# B&R Automation Studio project NAINV104C00R8L515F00 (part 11)

#### Act_OptP0200ToP0201AccDat.st
```iecst
ACTION Act_OptP0200ToP0201AccDat:

	//Control
	IF (tyP0200OpsGen.tyOps.tyBtnAccDat.bRtCompl = TRUE) OR (tyP0201OpsConv.tyOps.tyBtnAccDat.bRtCompl = TRUE) THEN
		tyP0200OpsGen.tyOps.tyBtnAccDat.bRtCompl	:= FALSE;
		tyP0201OpsConv.tyOps.tyBtnAccDat.bRtCompl	:= FALSE;

		bProdAccData	:= TRUE;
	END_IF

	//Button Appearance
	IF (p_bLFFollowerProdAccDataMnl = TRUE) OR (p_bUSHermesAccDataMnl = TRUE) OR (p_bLCSLFAccDataMnl = TRUE) THEN

		fbAccDatBlinkTm(IN := TRUE);

		IF fbAccDatBlinkTm.Q THEN
			fbAccDatBlinkTm(IN := FALSE);
			IF tyP0200OpsGen.tyOps.tyBitmapAccDat.usiValueIdx = 1 THEN
				tyP0200OpsGen.tyOps.tyBitmapAccDat.usiValueIdx		:= 0;
				tyP0201OpsConv.tyOps.tyBitmapAccDat.usiValueIdx	:= 0;
			ELSE
				tyP0200OpsGen.tyOps.tyBitmapAccDat.usiValueIdx		:= 1;
				tyP0201OpsConv.tyOps.tyBitmapAccDat.usiValueIdx	:= 1;
			END_IF
		END_IF

		fUIInRtStatOff(ADR(tyP0200OpsGen.tyOps.tyBtnAccDat.uiRtStat));
		fUIInRtStatOff(ADR(tyP0201OpsConv.tyOps.tyBtnAccDat.uiRtStat));

		fUIInRtStatOff(ADR(tyP0200OpsGen.tyOps.tyBitmapAccDat.uiRtStat));
		fUIInRtStatOff(ADR(tyP0201OpsConv.tyOps.tyBitmapAccDat.uiRtStat));

	ELSE

		fbAccDatBlinkTm(IN := FALSE);

		tyP0200OpsGen.tyOps.tyBitmapAccDat.usiValueIdx	:= 0;
		tyP0201OpsConv.tyOps.tyBitmapAccDat.usiValueIdx	:= 0;

		fUIInRtStatHide(ADR(tyP0200OpsGen.tyOps.tyBtnAccDat.uiRtStat));
		fUIInRtStatHide(ADR(tyP0201OpsConv.tyOps.tyBtnAccDat.uiRtStat));

		fUIInRtStatHide(ADR(tyP0200OpsGen.tyOps.tyBitmapAccDat.uiRtStat));
		fUIInRtStatHide(ADR(tyP0201OpsConv.tyOps.tyBitmapAccDat.uiRtStat));

	END_IF

//	IF p_tyNtParamCurr.bLFPrep THEN
//		IF p_bLFFollowerDSAllow=FALSE THEN
//			tyP0200OpsGen.tyOps.tyTxtLdrInActiveCtrl.usiValueIdx	:= 0;
//			tyP0201OpsConv.tyOps.tyTxtLdrInActiveCtrl.usiValueIdx	:= 0;
//
//			fUIInRtStatOff(ADR(tyP0200OpsGen.tyOps.tyTxtLdrInActiveCtrl.uiRtStat));
//			fUIInRtStatOff(ADR(tyP0201OpsConv.tyOps.tyTxtLdrInActiveCtrl.uiRtStat));
//			fUIInRtStatOff(ADR(tyP0200OpsGen.tyOps.tyBitmapWarningLF.uiRtStat));
//			fUIInRtStatOff(ADR(tyP0201OpsConv.tyOps.tyBitmapWarningLF.uiRtStat));
//
//		ELSIF p_bLFFollowerUSAllow=FALSE THEN
//			IF p_tyMcParamCurr.bSectionLeader THEN
//				tyP0200OpsGen.tyOps.tyTxtLdrInActiveCtrl.usiValueIdx	:= 3;
//				tyP0201OpsConv.tyOps.tyTxtLdrInActiveCtrl.usiValueIdx	:= 3;
//
//				fUIInRtStatOff(ADR(tyP0200OpsGen.tyOps.tyTxtLdrInActiveCtrl.uiRtStat));
//				fUIInRtStatOff(ADR(tyP0201OpsConv.tyOps.tyTxtLdrInActiveCtrl.uiRtStat));
//				fUIInRtStatOff(ADR(tyP0200OpsGen.tyOps.tyBitmapWarningLF.uiRtStat));
//				fUIInRtStatOff(ADR(tyP0201OpsConv.tyOps.tyBitmapWarningLF.uiRtStat));
//			ELSE
//				tyP0200OpsGen.tyOps.tyTxtLdrInActiveCtrl.usiValueIdx	:= 2;
//				tyP0201OpsConv.tyOps.tyTxtLdrInActiveCtrl.usiValueIdx	:= 2;
//
//				fUIInRtStatOff(ADR(tyP0200OpsGen.tyOps.tyTxtLdrInActiveCtrl.uiRtStat));
//				fUIInRtStatOff(ADR(tyP0201OpsConv.tyOps.tyTxtLdrInActiveCtrl.uiRtStat));
//				fUIInRtStatOff(ADR(tyP0200OpsGen.tyOps.tyBitmapWarningLF.uiRtStat));
//				fUIInRtStatOff(ADR(tyP0201OpsConv.tyOps.tyBitmapWarningLF.uiRtStat));
//			END_IF
//		ELSE
//			IF p_bLFFollowerLdrSeqCtrlInActive THEN
//				tyP0200OpsGen.tyOps.tyTxtLdrInActiveCtrl.usiValueIdx	:= 1;
//				tyP0201OpsConv.tyOps.tyTxtLdrInActiveCtrl.usiValueIdx	:= 1;
//
//				fUIInRtStatOff(ADR(tyP0200OpsGen.tyOps.tyTxtLdrInActiveCtrl.uiRtStat));
//				fUIInRtStatOff(ADR(tyP0201OpsConv.tyOps.tyTxtLdrInActiveCtrl.uiRtStat));
//				fUIInRtStatOff(ADR(tyP0200OpsGen.tyOps.tyBitmapWarningLF.uiRtStat));
//				fUIInRtStatOff(ADR(tyP0201OpsConv.tyOps.tyBitmapWarningLF.uiRtStat));
//			ELSE
//				fUIInRtStatHide(ADR(tyP0200OpsGen.tyOps.tyTxtLdrInActiveCtrl.uiRtStat));
//				fUIInRtStatHide(ADR(tyP0201OpsConv.tyOps.tyTxtLdrInActiveCtrl.uiRtStat));
//				fUIInRtStatHide(ADR(tyP0200OpsGen.tyOps.tyBitmapWarningLF.uiRtStat));
//				fUIInRtStatHide(ADR(tyP0201OpsConv.tyOps.tyBitmapWarningLF.uiRtStat));
//			END_IF
//		END_IF
//	ELSE
//		fUIInRtStatHide(ADR(tyP0200OpsGen.tyOps.tyTxtLdrInActiveCtrl.uiRtStat));
//		fUIInRtStatHide(ADR(tyP0201OpsConv.tyOps.tyTxtLdrInActiveCtrl.uiRtStat));
//		fUIInRtStatHide(ADR(tyP0200OpsGen.tyOps.tyBitmapWarningLF.uiRtStat));
//		fUIInRtStatHide(ADR(tyP0201OpsConv.tyOps.tyBitmapWarningLF.uiRtStat));
//	END_IF

END_ACTION
```

#### Act_OptP0200ToP0201BypsInitConv.st
```iecst
ACTION Act_OptP0200ToP0201BypsInitConv:

	IF p_tyNtParamCurr.bProjBypsInitConvPrep THEN

		(*Display*)
		//Initializing Conveyor
		IF EDGEPOS(p_bOpsInvertStepInitConv) THEN
			fUIInRtStatOff(ADR(tyP0200OpsGen.tyBypsInitConv.tyLyr.uiRtStat));
			fUIInRtStatOff(ADR(tyP0201OpsConv.tyBypsInitConv.tyLyr.uiRtStat));
		END_IF

		//Initializing Conveyor Done
		IF EDGENEG(p_bOpsInvertStepInitConv) THEN
			fUIInRtStatHide(ADR(tyP0200OpsGen.tyBypsInitConv.tyLyr.uiRtStat));
			fUIInRtStatHide(ADR(tyP0201OpsConv.tyBypsInitConv.tyLyr.uiRtStat));

			bOpsBypsInitConv	:= FALSE;
		END_IF

		//Blinking Button
		IF tyP0200OpsGen.tyBypsInitConv.tyLyr.uiRtStat.0 = FALSE THEN

			fbBypsInitConvBlinkTm(IN := TRUE);

			IF fbBypsInitConvBlinkTm.Q THEN
				fbBypsInitConvBlinkTm(IN := FALSE);

				IF tyP0200OpsGen.tyBypsInitConv.tyBtnBypsInitConv.usiBitmapIdx = 0 THEN
					tyP0200OpsGen.tyBypsInitConv.tyBtnBypsInitConv.usiBitmapIdx		:= 1;
					tyP0201OpsConv.tyBypsInitConv.tyBtnBypsInitConv.usiBitmapIdx	:= 1;

				ELSE
					tyP0200OpsGen.tyBypsInitConv.tyBtnBypsInitConv.usiBitmapIdx		:= 0;
					tyP0201OpsConv.tyBypsInitConv.tyBtnBypsInitConv.usiBitmapIdx	:= 0;
				END_IF

			END_IF

		ELSE

			fbBypsInitConvBlinkTm(IN := FALSE);

			tyP0200OpsGen.tyBypsInitConv.tyBtnBypsInitConv.usiBitmapIdx		:= 0;
			tyP0201OpsConv.tyBypsInitConv.tyBtnBypsInitConv.usiBitmapIdx	:= 0;
		END_IF

		(*Control*)
		IF tyP0200OpsGen.tyBypsInitConv.tyBtnBypsInitConv.bRtCompl OR tyP0201OpsConv.tyBypsInitConv.tyBtnBypsInitConv.bRtCompl THEN
			tyP0200OpsGen.tyBypsInitConv.tyBtnBypsInitConv.bRtCompl		:= FALSE;
			tyP0201OpsConv.tyBypsInitConv.tyBtnBypsInitConv.bRtCompl	:= FALSE;

			fUIInRtStatHide(ADR(tyP0200OpsGen.tyBypsInitConv.tyLyr.uiRtStat));
			fUIInRtStatHide(ADR(tyP0201OpsConv.tyBypsInitConv.tyLyr.uiRtStat));

			bOpsBypsInitConv	:= TRUE;

		ELSIF tyP0200OpsGen.tyBypsInitConv.tyHotspotClose.bRtCompl OR tyP0201OpsConv.tyBypsInitConv.tyHotspotClose.bRtCompl THEN
			tyP0200OpsGen.tyBypsInitConv.tyHotspotClose.bRtCompl	:= FALSE;
			tyP0201OpsConv.tyBypsInitConv.tyHotspotClose.bRtCompl	:= FALSE;

			fUIInRtStatHide(ADR(tyP0200OpsGen.tyBypsInitConv.tyLyr.uiRtStat));
			fUIInRtStatHide(ADR(tyP0201OpsConv.tyBypsInitConv.tyLyr.uiRtStat));

		END_IF

	END_IF

END_ACTION
```

#### Act_OptP0200ToP0201RlsNewProd.st
```iecst
ACTION Act_OptP0200ToP0201RlsNewProd:

	IF p_tyNtParamCurr.bProjRlsNewProdPrep = TRUE THEN

		//Control
		IF (tyP0200OpsGen.tyOps.tyBtnRlsNewProd.bRtCompl = TRUE) OR (tyP0201OpsConv.tyOps.tyBtnRlsNewProd.bRtCompl = TRUE) THEN
			tyP0200OpsGen.tyOps.tyBtnRlsNewProd.bRtCompl	:= FALSE;
			tyP0201OpsConv.tyOps.tyBtnRlsNewProd.bRtCompl	:= FALSE;

			bRlsNewProd	:= TRUE;
		END_IF

		//Button Appearance
		IF p_bOpsRun = TRUE AND  p_bFollower1WaitRlsProd = TRUE THEN
			fbRlsNewProdBlinkTm(IN := TRUE);

			IF fbRlsNewProdBlinkTm.Q THEN
				fbRlsNewProdBlinkTm(IN := FALSE);
				IF (tyP0200OpsGen.tyOps.tyBitmapRlsNewProd.usiValueIdx = 1) THEN
					tyP0200OpsGen.tyOps.tyBitmapRlsNewProd.usiValueIdx	:= 0;
					tyP0201OpsConv.tyOps.tyBitmapRlsNewProd.usiValueIdx	:= 0;
				ELSE
					tyP0200OpsGen.tyOps.tyBitmapRlsNewProd.usiValueIdx	:= 1;
					tyP0201OpsConv.tyOps.tyBitmapRlsNewProd.usiValueIdx	:= 1;
				END_IF
			END_IF

			fUIInRtStatOff(ADR(tyP0200OpsGen.tyOps.tyBtnRlsNewProd.uiRtStat));
			fUIInRtStatOff(ADR(tyP0201OpsConv.tyOps.tyBtnRlsNewProd.uiRtStat));

			fUIInRtStatOff(ADR(tyP0200OpsGen.tyOps.tyBitmapRlsNewProd.uiRtStat));
			fUIInRtStatOff(ADR(tyP0201OpsConv.tyOps.tyBitmapRlsNewProd.uiRtStat));

		ELSE
			bRlsNewProd	:= FALSE;

			fbRlsNewProdBlinkTm(IN := FALSE);

			tyP0200OpsGen.tyOps.tyBitmapRlsNewProd.usiValueIdx	:= 0;
			tyP0201OpsConv.tyOps.tyBitmapRlsNewProd.usiValueIdx	:= 0;

			fUIInRtStatHide(ADR(tyP0200OpsGen.tyOps.tyBtnRlsNewProd.uiRtStat));
			fUIInRtStatHide(ADR(tyP0201OpsConv.tyOps.tyBtnRlsNewProd.uiRtStat));

			fUIInRtStatHide(ADR(tyP0200OpsGen.tyOps.tyBitmapRlsNewProd.uiRtStat));
			fUIInRtStatHide(ADR(tyP0201OpsConv.tyOps.tyBitmapRlsNewProd.uiRtStat));

		END_IF

	ELSE

		bRlsNewProd	:= TRUE;

	END_IF

END_ACTION
```

#### Act_EntP0300Disp.st
```iecst
ACTION Act_EntP0300Disp:

	//Access Addres
	p_tyC0005Main ACCESS ADR(tyCommon.tyMain);

	p_tyC0007Notif ACCESS ADR(tyCommon.tyNotif);

	p_tyC0008MsgBox ACCESS ADR(tyP0300McInfo.tyMsgBoxHide);

	p_tyC0009Info ACCESS ADR(tyCommon.tyInfo);

	p_tyP0300McInfo ACCESS ADR(tyP0300McInfo.tyMcInfo);

	p_tyC0011Loading ACCESS ADR(tyCommon.tyLoading);

	//Display
	tyP0300McInfo.tyMcInfo.tyStringMcNm.sValue	:= p_tyMcParamCurr.sMcNm;

	fUIInRtStatHide(ADR(tyP0300McInfo.tyMcInfo.tyBtnPlaySong.uiRtStat));
	fUIInRtStatHide(ADR(tyP0300McInfo.tyMcInfo.tyDrpDnSong.uiRtStat));

END_ACTION
```

#### Act_OptP0300Songt.st
```iecst
ACTION Act_OptP0300Song:

	IF EDGENEG(bSongEn) THEN
		tyP0300McInfo.tyMcInfo.tyBtnPlaySong.bValue := FALSE;
	ELSE
		bSongEn := tyP0300McInfo.tyMcInfo.tyBtnPlaySong.bValue;
	END_IF

	uiSongIndex := USINT_TO_UINT(tyP0300McInfo.tyMcInfo.tyDrpDnSong.usiValueIdx);

END_ACTION
```

#### Act_EntP0400Disp.st
```iecst
ACTION Act_EntP0400Disp:

	//Access Addres
	p_tyC0005Main ACCESS ADR(tyCommon.tyMain);

	p_tyC0007Notif ACCESS ADR(tyCommon.tyNotif);

	p_tyC0008MsgBox ACCESS ADR(tyP0400ProdSel.tyMsgBoxHide);

	p_tyC0009Info ACCESS ADR(tyCommon.tyInfo);

	p_tyC0011Loading ACCESS ADR(tyCommon.tyLoading);

	p_tyC0012RcpPopUp ACCESS ADR(tyP0400ProdSel.tyRcpPopUp);

	p_tyP0400ProdSel ACCESS ADR(tyP0400ProdSel.tyProdSel);
	p_tyP0400RcpDet ACCESS ADR(tyP0400ProdSel.tyRcpDet);

	//Display
	tyP1040ProdSet.tyProdSet.tyBtnSort.bRtCompl			:= FALSE;
	tyP1040ProdSet.tyProdSet.tyBtnSort.bValue			:= FALSE;
	tyP0400ProdSel.tyProdSel.tyStringSearch.bRtCompl	:= TRUE;
	tyP0400ProdSel.tyProdSel.tyStringSearch.sValue		:= '';
	fUIInRtStatHide(ADR(tyP0400ProdSel.tyRcpDet.tyLyr.uiRtStat));

	fUIInRtStatHide(ADR(tyP0400ProdSel.tyRcpPopUp.tyLyr.uiRtStat)); // Hide Pop Up Layer

	//Product Selection
	tyP0400ProdSel.tyProdSel.tyStringRecipeNm.sValue		:= p_tyProdRcpCurrRcp0.sRcpNm;
	tyP0400ProdSel.tyProdSel.tyNumProdWidth.diValue			:= p_tyProdRcpCurrRcp0.diWidthInUM;
	tyP0400ProdSel.tyProdSel.tyNumProdWidth2.diValue	:= p_tyProdRcpCurrRcp0.diWidthInUM2;
	tyP0400ProdSel.tyProdSel.tyTxtMcMod.usiValueIdx			:= p_tyProdRcpCurrRcp0.usiMcMod;
	tyP0400ProdSel.tyProdSel.tyTxtFlippedBrd.usiValueIdx	:= p_tyProdRcpCurrRcp0.usiFlippedBrd;
	tyP0400ProdSel.tyProdSel.tyStringMatchCode.sValue		:= p_tyProdRcpCurrRcp0.sMatchCode;

END_ACTION
```

#### Act_OptP0400Mask.st
```iecst
ACTION Act_OptP0400Mask:

	IF p_tyNtParamCurr.bLCSLFPrep AND p_tyMcParamCurr.bLCSLFEn THEN
		tyP0400ProdSel.tyProdSel.tyBtnLoad.uiMaskRtStat.0	:= FALSE;
	ELSE
		tyP0400ProdSel.tyProdSel.tyBtnLoad.uiMaskRtStat.0	:= (tyP0400ProdSel.tyProdSel.tyTableRecipe.a_tyStringDataCol1[tyP0400Table.uiSelectedRow].sValue <> '') AND (tyP0400ProdSel.tyProdSel.tyStringSearch.bRtCompl = FALSE);
	END_IF

	tyP0400ProdSel.tyProdSel.tyBtnPreview.uiMaskRtStat.0	:= (tyP0400ProdSel.tyProdSel.tyTableRecipe.a_tyStringDataCol1[tyP0400Table.uiSelectedRow].sValue <> '') AND (tyP0400ProdSel.tyProdSel.tyStringSearch.bRtCompl = FALSE) AND (tyP0400ProdSel.tyProdSel.tyBtnLoad.bRtCompl = FALSE);

	tyP0400ProdSel.tyProdSel.tyBtnSort.uiMaskRtStat.0		:= (tyP0400ProdSel.tyProdSel.tyTableRecipe.a_tyStringDataCol1[1].sValue <> '') AND (tyP0400ProdSel.tyProdSel.tyStringSearch.bRtCompl = FALSE) AND (tyP0400ProdSel.tyProdSel.tyBtnLoad.bRtCompl = FALSE);

END_ACTION
```

#### Act_OptP0400Search.st
```iecst
ACTION Act_OptP0400Search:

	IF tyP0400ProdSel.tyProdSel.tyStringSearch.bRtCompl = TRUE THEN	//Search Input Valid
		IF tyP0400ProdSel.tyProdSel.tyStringSearch.sValue = '' THEN
			FOR i := 1 TO c_uiP0400TableSize DO
				tyP0400ProdSel.tyProdSel.tyTableRecipe.a_tyStringDataCol0[i].sValue	:= UINT_TO_STRING(tyP0400Table.uiTablePos + i - 1);
				tyP0400ProdSel.tyProdSel.tyTableRecipe.a_tyStringDataCol1[i].sValue	:= p_tyProdRcpCurrList[tyP0400Table.uiTablePos + i - 1].sRcpNm;
				tyP0400ProdSel.tyProdSel.tyTableRecipe.a_tyStringDataCol2[i].sValue	:= p_tyProdRcpCurrList[tyP0400Table.uiTablePos + i - 1].sDisplayInfo;
			END_FOR

			tyP0400ProdSel.tyProdSel.tyStringSearch.bRtCompl	:= FALSE;

			IF tyP0400ProdSel.tyProdSel.tyBtnSort.bValue THEN
				bFilterSortP0400	:= TRUE;
			END_IF

		ELSE
			//Mask
			tyP0400ProdSel.tyProdSel.tyTableRecipe.uiMaskRtStat.0	:= FALSE;

			sProdRcpSearch	:= tyP0400ProdSel.tyProdSel.tyStringSearch.sValue;

			eProdRcpAct	:= ProdRcpActFilter;

			IF p_eProdRcpStat = ProdRcpActFilter AND p_eProdRcpStatus = Done THEN
				eProdRcpAct		:= ProdRcpActIdle;

				FOR i := 1 TO c_uiP0400TableSize DO
					tyP0400ProdSel.tyProdSel.tyTableRecipe.a_tyStringDataCol0[i].sValue	:= UINT_TO_STRING(tyP0400Table.uiTablePos + i - 1);
					tyP0400ProdSel.tyProdSel.tyTableRecipe.a_tyStringDataCol1[i].sValue	:= p_tyProdRcpFilterList[tyP0400Table.uiTablePos + i - 1].sRcpNm;
					tyP0400ProdSel.tyProdSel.tyTableRecipe.a_tyStringDataCol2[i].sValue	:= p_tyProdRcpFilterList[tyP0400Table.uiTablePos + i - 1].sDisplayInfo;
				END_FOR

				//Unmask
				tyP0400ProdSel.tyProdSel.tyTableRecipe.uiMaskRtStat.0	:= TRUE;

				tyP0400ProdSel.tyProdSel.tyStringSearch.bRtCompl		:= FALSE;

				IF tyP0400ProdSel.tyProdSel.tyBtnSort.bValue THEN
					bFilterSortP0400	:= TRUE;
				END_IF

			ELSIF p_eProdRcpStatus = Error THEN
				FOR i := 1 TO c_uiP0400TableSize DO
					tyP0400ProdSel.tyProdSel.tyTableRecipe.a_tyStringDataCol0[i].sValue		:= UINT_TO_STRING(tyP0400Table.uiTablePos + i - 1);
					tyP0400ProdSel.tyProdSel.tyTableRecipe.a_tyStringDataCol1[i].sValue		:= '';
					tyP0400ProdSel.tyProdSel.tyTableRecipe.a_tyStringDataCol2[i].sValue		:= '';
				END_FOR

				p_tyC0008MsgBox ACCESS ADR (tyP0400ProdSel.tyMsgBoxListErr);

				IF tyP0400ProdSel.tyMsgBoxListErr.tyBtnNo.bRtCompl = TRUE THEN
					tyP0400ProdSel.tyMsgBoxListErr.tyBtnNo.bRtCompl 		:= TRUE;
					tyP0400ProdSel.tyMsgBoxListErr.tyBtnNo.bValue			:= TRUE;

					p_tyC0008MsgBox ACCESS ADR (tyP0400ProdSel.tyMsgBoxHide);

					//Unmask
					tyP0400ProdSel.tyProdSel.tyTableRecipe.uiMaskRtStat.0	:= TRUE;

					//Reset
					tyP0400ProdSel.tyProdSel.tyStringSearch.bRtCompl		:= FALSE;
				END_IF
			END_IF
		END_IF
	END_IF

END_ACTION
```

#### Act_OptP0400Load.st
```iecst
ACTION Act_OptP0400Load:

	IF tyP0400ProdSel.tyProdSel.tyBtnLoad.bRtCompl = TRUE THEN

		IF usiSelProdRcpStep = 0 THEN
			//Message Confirmation Ask - Load Product Recipe
			//Mask
			tyP0400ProdSel.tyProdSel.tyTableRecipe.uiMaskRtStat		:= FALSE;
			tyP0400ProdSel.tyProdSel.tyStringSearch.uiMaskRtStat	:= FALSE;

			p_tyC0008MsgBox ACCESS ADR(tyP0400ProdSel.tyMsgBoxSelRcpAsk);

			IF tyP0400ProdSel.tyMsgBoxSelRcpAsk.tyBtnYes.bRtCompl = TRUE THEN
				tyP0400ProdSel.tyMsgBoxSelRcpAsk.tyBtnYes.bRtCompl	:= FALSE;
				tyP0400ProdSel.tyMsgBoxSelRcpAsk.tyBtnYes.bValue	:= FALSE;

				p_tyC0008MsgBox ACCESS ADR(tyP0400ProdSel.tyMsgBoxHide);

				usiSelProdRcpStep	:= 1;

			ELSIF tyP0400ProdSel.tyMsgBoxSelRcpAsk.tyBtnNo.bRtCompl = TRUE THEN
				tyP0400ProdSel.tyMsgBoxSelRcpAsk.tyBtnNo.bRtCompl	:= FALSE;
				tyP0400ProdSel.tyMsgBoxSelRcpAsk.tyBtnNo.bValue		:= FALSE;

				p_tyC0008MsgBox ACCESS ADR(tyP0400ProdSel.tyMsgBoxHide);

				usiSelProdRcpStep	:= 99;

			END_IF

		ELSIF usiSelProdRcpStep = 1 THEN
			//Load Product Recipe
			tyProdRcpInfoIn.sRcpNm	:= tyP0400ProdSel.tyProdSel.tyTableRecipe.a_tyStringDataCol1[tyP0400Table.uiSelectedRow].sValue;

			eProdRcpAct	:= ProdRcpActLoadRcp;

			IF p_eProdRcpStat = ProdRcpActLoadRcp AND p_eProdRcpStatus = Done THEN
				eProdRcpAct	:= ProdRcpActIdle;

				IF p_bProdRcpNmEmpty = TRUE AND p_bProdRcpNmNotExist = TRUE THEN
					usiSelProdRcpStep	:= 2;
				ELSE
					//Update UI Current Recipe
					tyP0400ProdSel.tyProdSel.tyStringRecipeNm.sValue	:= p_tyProdRcpCurrRcp0.sRcpNm;
					tyP0400ProdSel.tyProdSel.tyNumProdWidth.diValue		:= p_tyProdRcpCurrRcp0.diWidthInUM;
					tyP0400ProdSel.tyProdSel.tyNumProdWidth2.diValue	:= p_tyProdRcpCurrRcp0.diWidthInUM2;
					tyP0400ProdSel.tyProdSel.tyTxtMcMod.usiValueIdx		:= p_tyProdRcpCurrRcp0.usiMcMod;
					tyP0400ProdSel.tyProdSel.tyTxtFlippedBrd.usiValueIdx:= p_tyProdRcpCurrRcp0.usiFlippedBrd;
					tyP0400ProdSel.tyProdSel.tyStringMatchCode.sValue	:= p_tyProdRcpCurrRcp0.sMatchCode;

					tyProdRcpCurrRcpWr	:= p_tyProdRcpCurrRcp0;

					IF ((NOT p_tyNtParamCurr.bLFUsrSetPrep AND p_tyNtParamCurr.bLeaderMc) OR (p_tyNtParamCurr.bLFUsrSetPrep AND p_tyMcParamCurr.bLFLeaderMc)) AND p_tyNtParamCurr.bLFPrep AND p_tyMcParamCurr.bLFEn AND p_tyUsrMgmtCurrAccessRgt.bLFCtrl THEN
						usiSelProdRcpStep	:= 98;
					ELSE
						usiSelProdRcpStep	:= 99;
					END_IF

				END_IF

			ELSIF p_eProdRcpStatus = Error THEN

				usiSelProdRcpStep	:= 99;

			END_IF

		ELSIF usiSelProdRcpStep = 2 THEN
			//Message Name Not Found
			p_tyC0008MsgBox ACCESS ADR(tyP0400ProdSel.tyMsgBoxSelRcpNoNm);

			IF tyP0400ProdSel.tyMsgBoxSelRcpNoNm.tyBtnNo.bRtCompl = TRUE THEN
				tyP0400ProdSel.tyMsgBoxSelRcpNoNm.tyBtnNo.bRtCompl	:= FALSE;
				tyP0400ProdSel.tyMsgBoxSelRcpNoNm.tyBtnNo.bValue	:= FALSE;

				p_tyC0008MsgBox ACCESS ADR(tyP0400ProdSel.tyMsgBoxHide);

				usiSelProdRcpStep	:= 99;

			END_IF

		ELSIF usiSelProdRcpStep = 98 THEN
			//Message Confirmation Ask - Go To Leader Follower Control Page
			p_tyC0008MsgBox ACCESS ADR(tyP0400ProdSel.tyMsgBoxGoToLFCtrlAsk);

			IF tyP0400ProdSel.tyMsgBoxGoToLFCtrlAsk.tyBtnYes.bRtCompl = TRUE THEN
				tyP0400ProdSel.tyMsgBoxGoToLFCtrlAsk.tyBtnYes.bRtCompl	:= FALSE;
				tyP0400ProdSel.tyMsgBoxGoToLFCtrlAsk.tyBtnYes.bValue	:= FALSE;

				p_tyC0008MsgBox ACCESS ADR(tyP0400ProdSel.tyMsgBoxHide);

				//Change Page
				eChgPage	:= UIP0700LFCtrl;

				//Start Operation
				tyCommon.tyMain.tyBtnStart.bRtCompl	:= TRUE;

				//Complete
				//Unmask
				tyP0400ProdSel.tyProdSel.tyTableRecipe.uiMaskRtStat		:= TRUE;
				tyP0400ProdSel.tyProdSel.tyStringSearch.uiMaskRtStat	:= TRUE;

				//Reset
				tyP0400ProdSel.tyProdSel.tyBtnLoad.bRtCompl	:= FALSE;
				tyP0400ProdSel.tyProdSel.tyBtnLoad.bValue	:= FALSE;

				usiSelProdRcpStep	:= 0;

			ELSIF tyP0400ProdSel.tyMsgBoxGoToLFCtrlAsk.tyBtnNo.bRtCompl = TRUE THEN
				tyP0400ProdSel.tyMsgBoxGoToLFCtrlAsk.tyBtnNo.bRtCompl	:= FALSE;
				tyP0400ProdSel.tyMsgBoxGoToLFCtrlAsk.tyBtnNo.bValue		:= FALSE;

				p_tyC0008MsgBox ACCESS ADR(tyP0400ProdSel.tyMsgBoxHide);

				usiSelProdRcpStep	:= 99;

			END_IF

		ELSIF usiSelProdRcpStep = 99 THEN
			//Complete
			//Unmask
			tyP0400ProdSel.tyProdSel.tyTableRecipe.uiMaskRtStat		:= TRUE;
			tyP0400ProdSel.tyProdSel.tyStringSearch.uiMaskRtStat	:= TRUE;

			//Reset
			tyP0400ProdSel.tyProdSel.tyBtnLoad.bRtCompl	:= FALSE;
			tyP0400ProdSel.tyProdSel.tyBtnLoad.bValue	:= FALSE;

			usiSelProdRcpStep	:= 0;

		END_IF

	END_IF

END_ACTION
```

#### Act_OptP0400Preview.st
```iecst
ACTION Act_OptP0400Preview:

	IF tyP0400ProdSel.tyProdSel.tyBtnPreview.bRtCompl = TRUE THEN

		tyProdRcpInfoIn.sRcpNm	:= tyP0400ProdSel.tyProdSel.tyTableRecipe.a_tyStringDataCol1[tyP0400Table.uiSelectedRow].sValue;

		eProdRcpAct	:= ProdRcpActGetInfo;

		IF	p_eProdRcpStat = ProdRcpActGetInfo AND p_eProdRcpStatus = Done THEN
			eProdRcpAct	:= ProdRcpActIdle;

			IF p_bProdRcpNmEmpty = TRUE AND p_bProdRcpNmNotExist = TRUE THEN
				tyP0400ProdSel.tyRcpDet.tyStringRecipeNm.sValue		:= '';
				tyP0400ProdSel.tyRcpDet.tyNumProdWidth.diValue		:= 100000;
				tyP0400ProdSel.tyRcpDet.tyNumProdWidth2.diValue		:= 100000;
				tyP0400ProdSel.tyRcpDet.tyTxtMcMod.usiValueIdx		:= p_tyMcParamCurr.usiDefaultMcMod;
				tyP0400ProdSel.tyRcpDet.tyTxtFlippedBrd.usiValueIdx	:= p_tyMcParamCurr.usiDefaultFlippedBrd;
				tyP0400ProdSel.tyRcpDet.tyStringMatchCode.sValue	:= '';
			ELSE
				tyP0400ProdSel.tyRcpDet.tyStringRecipeNm.sValue		:= p_tyProdRcpInfoOut.sRcpNm;
				tyP0400ProdSel.tyRcpDet.tyNumProdWidth.diValue		:= p_tyProdRcpInfoOut.diWidthInUM;
				tyP0400ProdSel.tyRcpDet.tyNumProdWidth2.diValue		:= p_tyProdRcpInfoOut.diWidthInUM2;
				tyP0400ProdSel.tyRcpDet.tyTxtMcMod.usiValueIdx		:= p_tyProdRcpInfoOut.usiMcMod;
				tyP0400ProdSel.tyRcpDet.tyTxtFlippedBrd.usiValueIdx	:= p_tyProdRcpInfoOut.usiFlippedBrd;
				tyP0400ProdSel.tyRcpDet.tyStringMatchCode.sValue	:= p_tyProdRcpInfoOut.sMatchCode;
			END_IF

			fUIInRtStatOff(ADR(tyP0400ProdSel.tyRcpDet.tyLyr.uiRtStat));

			tyP0400ProdSel.tyProdSel.tyBtnPreview.bRtCompl	:= FALSE;

		END_IF

	END_IF

	IF tyP0400ProdSel.tyRcpDet.tyHotspotClose.bRtCompl = TRUE THEN
		tyP0400ProdSel.tyRcpDet.tyHotspotClose.bRtCompl	:= FALSE;
		tyP0400ProdSel.tyProdSel.tyBtnPreview.bValue	:= FALSE;

		//Hide Recipe Details
		fUIInRtStatHide(ADR(tyP0400ProdSel.tyRcpDet.tyLyr.uiRtStat));

	END_IF

	//254 Characters are Shown
	IF tyP0400ProdSel.tyRcpDet.tyHotspotShowLRcp.bRtCompl = TRUE THEN
		tyP0400ProdSel.tyRcpDet.tyHotspotShowLRcp.bRtCompl  := FALSE;

		fUIInRtStatOff(ADR(tyP0400ProdSel.tyRcpPopUp.tyLyr.uiRtStat));

		tyP0400ProdSel.tyRcpPopUp.tyStringInfo.sValue  :=  tyP0400ProdSel.tyProdSel.tyTableRecipe.a_tyStringDataCol1[tyP0400Table.uiSelectedRow].sValue; // Show 254 Characters

	ELSIF tyP0400ProdSel.tyRcpPopUp.tyHotspotClose.bRtCompl = TRUE THEN
		tyP0400ProdSel.tyRcpPopUp.tyHotspotClose.bRtCompl := FALSE;

		fUIInRtStatHide(ADR(tyP0400ProdSel.tyRcpPopUp.tyLyr.uiRtStat)); // Hide Pop Up Again

	END_IF

END_ACTION
```

#### Act_OptP0400Table.st
```iecst
ACTION Act_OptP0400Table:

	//Call Table FB
	fbP0400Table.sVisuNm			:= tyP0400Table.sVisuNm;
	fbP0400Table.udiWorkAreaStartX	:= 359;
	fbP0400Table.udiWorkAreaEndX	:= 770;
	fbP0400Table.udiWorkAreaStartY	:= 93;
	fbP0400Table.udiWorkAreaEndY	:= 415;
	fbP0400Table.udiMinXDist		:= 20;
	fbP0400Table.udiMinYDist		:= 20;
	fbP0400Table.uiSlideScale		:= c_uiP0400TableSize;
	fbP0400Table.iTotalData			:= UDINT_TO_INT(c_udiProdRcpMax);;
	fbP0400Table.iTotalRow			:= c_uiP0400TableSize;
	fbP0400Table(uiSliderStatus := tyP0400ProdSel.tyProdSel.tyTableRecipe.tyUISlider.uiRtStat , a_tyUIHotspot := tyP0400ProdSel.tyProdSel.tyTableRecipe.a_tyHotspot , uiTablePos := tyP0400Table.uiTablePos , iSliderPos := tyP0400ProdSel.tyProdSel.tyTableRecipe.tyUISlider.iValue);

	tyP0400Table.uiSelectedRow		:= fbP0400Table.uiSelectedRow;
	tyP0400Table.bTableActive		:= fbP0400Table.bTableActive;
	tyP0400Table.bSliderActive		:= fbP0400Table.bSliderActive;

	//Table Content

	IF tyP0400Table.bTableActive = TRUE OR tyP0400Table.bSliderActive = TRUE OR bUpdateP0400Table THEN
		FOR i := 1 TO c_uiP0400TableSize DO
			IF tyP0400ProdSel.tyProdSel.tyBtnSort.bValue THEN

				tyP0400ProdSel.tyProdSel.tyTableRecipe.a_tyStringDataCol0[i].sValue	:= UINT_TO_STRING(tyP0400Table.uiTablePos + i - 1);
				tyP0400ProdSel.tyProdSel.tyTableRecipe.a_tyStringDataCol1[i].sValue	:= p_tyProdRcpSortedList[tyP0400Table.uiTablePos + i - 1].sRcpNm;
				tyP0400ProdSel.tyProdSel.tyTableRecipe.a_tyStringDataCol2[i].sValue	:= p_tyProdRcpSortedList[tyP0400Table.uiTablePos + i - 1].sDisplayInfo;

			ELSE

			IF tyP0400ProdSel.tyProdSel.tyStringSearch.sValue = '' THEN
				tyP0400ProdSel.tyProdSel.tyTableRecipe.a_tyStringDataCol0[i].sValue	:= UINT_TO_STRING(tyP0400Table.uiTablePos + i - 1);
				tyP0400ProdSel.tyProdSel.tyTableRecipe.a_tyStringDataCol1[i].sValue	:= p_tyProdRcpCurrList[tyP0400Table.uiTablePos + i - 1].sRcpNm;
				tyP0400ProdSel.tyProdSel.tyTableRecipe.a_tyStringDataCol2[i].sValue	:= p_tyProdRcpCurrList[tyP0400Table.uiTablePos + i - 1].sDisplayInfo;
			ELSE
				tyP0400ProdSel.tyProdSel.tyTableRecipe.a_tyStringDataCol0[i].sValue	:= UINT_TO_STRING(tyP0400Table.uiTablePos + i - 1);
				tyP0400ProdSel.tyProdSel.tyTableRecipe.a_tyStringDataCol1[i].sValue	:= p_tyProdRcpFilterList[tyP0400Table.uiTablePos + i - 1].sRcpNm;
				tyP0400ProdSel.tyProdSel.tyTableRecipe.a_tyStringDataCol2[i].sValue	:= p_tyProdRcpFilterList[tyP0400Table.uiTablePos + i - 1].sDisplayInfo;
				END_IF

			END_IF
		END_FOR

		IF bUpdateP0400Table THEN
			bUpdateP0400Table := FALSE;
		END_IF

	END_IF

	//Selected Row
	IF tyP0400Table.uiSelectedRow <> tyP0400Table.uiSelectedRowOld THEN
		FOR i := 1 TO c_uiP0400TableSize DO
			IF tyP0400Table.uiSelectedRow = i THEN
				tyP0400ProdSel.tyProdSel.tyTableRecipe.a_tyStringDataCol1[i].usiColor	:= 1;
				tyP0400ProdSel.tyProdSel.tyTableRecipe.a_tyStringDataCol2[i].usiColor	:= 1;
			ELSE
				tyP0400ProdSel.tyProdSel.tyTableRecipe.a_tyStringDataCol1[i].usiColor	:= 0;
				tyP0400ProdSel.tyProdSel.tyTableRecipe.a_tyStringDataCol2[i].usiColor	:= 0;
			END_IF
		END_FOR

		tyP0400Table.uiSelectedRowOld	:= tyP0400Table.uiSelectedRow;
	END_IF

END_ACTION
```

#### Act_OptP0400Sort.st
```iecst
ACTION Act_OptP0400Sort:

	IF tyP0400ProdSel.tyProdSel.tyBtnSort.bValue THEN
		tyP0400ProdSel.tyProdSel.tyBtnSort.usiTxtIdx 	:= 1;
	ELSE
		tyP0400ProdSel.tyProdSel.tyBtnSort.usiTxtIdx 	:= 0;
	END_IF

	IF tyP0400ProdSel.tyProdSel.tyBtnSort.bRtCompl OR (bFilterSortP0400 AND p_eProdRcpStat<> ProdRcpActFilter) THEN

		IF tyP0400ProdSel.tyProdSel.tyBtnSort.bValue THEN

			tyP0400ProdSel.tyProdSel.tyTableRecipe.uiMaskRtStat.0	:= FALSE;

			sProdRcpSearch	:= tyP0400ProdSel.tyProdSel.tyStringSearch.sValue;

			eProdRcpAct	:= ProdRcpActSort;

			IF p_eProdRcpStat = ProdRcpActSort AND p_eProdRcpStatus = Done THEN
				eProdRcpAct		:= ProdRcpActIdle;

				FOR i := 1 TO c_uiP1040TableSize DO
					tyP0400ProdSel.tyProdSel.tyTableRecipe.a_tyStringDataCol0[i].sValue	:= UINT_TO_STRING(tyP0400Table.uiTablePos + i - 1);
					tyP0400ProdSel.tyProdSel.tyTableRecipe.a_tyStringDataCol1[i].sValue	:= p_tyProdRcpSortedList[tyP0400Table.uiTablePos + i - 1].sRcpNm;
					tyP0400ProdSel.tyProdSel.tyTableRecipe.a_tyStringDataCol2[i].sValue	:= p_tyProdRcpSortedList[tyP0400Table.uiTablePos + i - 1].sDisplayInfo;
				END_FOR

				bFilterSortP0400	:= FALSE;

				//Unmask
				tyP0400ProdSel.tyProdSel.tyTableRecipe.uiMaskRtStat.0	:= TRUE;

				tyP0400ProdSel.tyProdSel.tyBtnSort.bRtCompl := FALSE;

			ELSIF p_eProdRcpStatus = Error THEN
				FOR i := 1 TO c_uiP0400TableSize DO
					tyP0400ProdSel.tyProdSel.tyTableRecipe.a_tyStringDataCol0[i].sValue		:= UINT_TO_STRING(tyP0400Table.uiTablePos + i - 1);
					tyP0400ProdSel.tyProdSel.tyTableRecipe.a_tyStringDataCol1[i].sValue		:= '';
					tyP0400ProdSel.tyProdSel.tyTableRecipe.a_tyStringDataCol2[i].sValue		:= '';
				END_FOR

				p_tyC0008MsgBox ACCESS ADR (tyP0400ProdSel.tyMsgBoxListErr);

				bFilterSortP0400	:= FALSE;

				IF tyP0400ProdSel.tyMsgBoxListErr.tyBtnNo.bRtCompl = TRUE THEN
					tyP0400ProdSel.tyMsgBoxListErr.tyBtnNo.bRtCompl 		:= TRUE;
					tyP0400ProdSel.tyMsgBoxListErr.tyBtnNo.bValue			:= TRUE;

					p_tyC0008MsgBox ACCESS ADR (tyP0400ProdSel.tyMsgBoxHide);

					//Unmask
					tyP0400ProdSel.tyProdSel.tyTableRecipe.uiMaskRtStat.0	:= TRUE;

					//Reset
					tyP0400ProdSel.tyProdSel.tyBtnSort.bRtCompl := FALSE;
				END_IF
			END_IF

		ELSE

			bUpdateP0400Table	:= TRUE;

			tyP0400ProdSel.tyProdSel.tyBtnSort.bRtCompl := FALSE;

		END_IF

	END_IF

END_ACTION
```

#### Act_OptP0400Keypad.st
```iecst
ACTION Act_OptP0400Keypad:

	IF fUIOutRtStatTPIsOpen(ADR(tyP0400ProdSel.tyProdSel.tyStringSearch.uiRtStat)) THEN
		tyProperty.tyKeypad.tyTxtTitle.sTxt	:= tyP0400ProdSel.tyProdSel.tyStringSearch.sKeypadTitle;

	END_IF

END_ACTION
```

#### Act_OptP0400RcpPopUp.st
```iecst
ACTION Act_OptP0400RcpPopUp:

	tyP0400ProdSel.tyProdSel.tyHotspotShowLRcp.uiRtStat.0	:= NOT(tyP0400ProdSel.tyProdSel.tyStringRecipeNm.sValue <> '');

	IF tyP0400ProdSel.tyProdSel.tyHotspotShowLRcp.bRtCompl = TRUE THEN
		tyP0400ProdSel.tyProdSel.tyHotspotShowLRcp.bRtCompl  := FALSE;

		fUIInRtStatOff(ADR(tyP0400ProdSel.tyRcpPopUp.tyLyr.uiRtStat));

		tyP0400ProdSel.tyRcpPopUp.tyStringInfo.sValue  :=  tyP0400ProdSel.tyProdSel.tyStringRecipeNm.sValue; // Show 254 Characters

	ELSIF tyP0400ProdSel.tyRcpPopUp.tyHotspotClose.bRtCompl = TRUE THEN
		tyP0400ProdSel.tyRcpPopUp.tyHotspotClose.bRtCompl := FALSE;

		fUIInRtStatHide(ADR(tyP0400ProdSel.tyRcpPopUp.tyLyr.uiRtStat)); // Hide Pop Up Again

	END_IF

END_ACTION
```

#### Act_EntP0600Disp.st
```iecst
ACTION Act_EntP0600Disp:

	//Access Addres
	p_tyC0005Main ACCESS ADR(tyCommon.tyMain);

	p_tyC0007Notif ACCESS ADR(tyCommon.tyNotif);

	p_tyC0008MsgBox ACCESS ADR(tyP0600Alm.tyMsgBoxHide);

	p_tyC0009Info ACCESS ADR(tyCommon.tyInfo);

	p_tyC0010RcyMsg ACCESS ADR(tyP0600Alm.tyRcyMsgHide);

	p_tyC0011Loading ACCESS ADR(tyCommon.tyLoading);

	p_tyP0600Alm ACCESS ADR(tyP0600Alm.tyAlm);

	tyP0600Alm.tyAlm.tyBtnCurr.bRtCompl := TRUE;

	//Reset
	bTeachStopperAtLftPos	:= FALSE;
	bTeachStopperAtRgtPos	:= FALSE;

END_ACTION
```

#### Act_OptP0600Alm.st
```iecst
ACTION Act_OptP0600Alm:

	IF tyP0600Alm.tyAlm.tyBtnHistory.bRtCompl = TRUE THEN
		tyP0600Alm.tyAlm.tyBtnHistory.bRtCompl		:= FALSE;
		tyP0600Alm.tyAlm.tyBtnHistory.bValue		:= TRUE;
		tyP0600Alm.tyAlm.tyBtnCurr.bValue			:= FALSE;
	ELSIF tyP0600Alm.tyAlm.tyBtnCurr.bRtCompl = TRUE THEN
		tyP0600Alm.tyAlm.tyBtnCurr.bRtCompl			:= FALSE;
		tyP0600Alm.tyAlm.tyBtnCurr.bValue			:= TRUE;
		tyP0600Alm.tyAlm.tyBtnHistory.bValue		:= FALSE;
	END_IF

	IF NOT p_bAlarmErr THEN
		memset(ADR(tyUIAlmData.bAlm) , 0 , SIZEOF(tyUIAlmData.bAlm));
	END_IF

	IF NOT p_bAlarmWarning THEN
		memset(ADR(tyUIAlmData.bWarning) , 0 , SIZEOF(tyUIAlmData.bWarning));
	ELSE
		IF (p_bUSHermesConnected) OR p_tyMcParamCurr.eUSComm = McSetCommModSMEMA THEN
			tyUIAlmData.bWarning[3114] := FALSE;
		END_IF
		IF (p_bDSHermesConnected) OR p_tyMcParamCurr.eDSComm = McSetCommModSMEMA THEN
			tyUIAlmData.bWarning[3363] := FALSE;
		END_IF
	END_IF

	IF tyP0600Alm.tyAlm.tyBtnCurr.bValue = TRUE THEN

		fUIInRtStatOff(ADR(tyP0600Alm.tyAlm.tyAlarm.tyUIAlmCur.uiRtStat));
		fUIInRtStatHide(ADR(tyP0600Alm.tyAlm.tyAlarm.tyUIAlmHis.uiRtStat));
		tyP0600Alm.tyAlm.tyBtnHistoryUp.uiMaskRtStat.0 		:= FALSE;
		tyP0600Alm.tyAlm.tyBtnHistoryDown.uiMaskRtStat.0 	:= FALSE;

		FOR i := 1 TO c_uiP0600TableSize DO
			IF p_bStartupUISettingsLoadDone THEN
				IF p_tyAlarmCurrList[i].eSeverity = AlmSeverityError THEN
					tyUIAlmData.bAlm[p_tyAlarmCurrList[i].udiErrorCode] := p_tyAlarmCurrList[i].bAlm;
				ELSIF p_tyAlarmCurrList[i].eSeverity = AlmSeverityWarning THEN
					tyUIAlmData.bWarning[p_tyAlarmCurrList[i].udiErrorCode] := p_tyAlarmCurrList[i].bWarning;
				END_IF
			END_IF
		END_FOR

	ELSIF tyP0600Alm.tyAlm.tyBtnHistory.bValue = TRUE THEN

		fUIInRtStatHide(ADR(tyP0600Alm.tyAlm.tyAlarm.tyUIAlmCur.uiRtStat));
		fUIInRtStatOff(ADR(tyP0600Alm.tyAlm.tyAlarm.tyUIAlmHis.uiRtStat));
		tyP0600Alm.tyAlm.tyBtnHistoryUp.uiMaskRtStat.0 		:= TRUE;
		tyP0600Alm.tyAlm.tyBtnHistoryDown.uiMaskRtStat.0 	:= TRUE;

	END_IF

END_ACTION
```

#### Act_OptP0600RcyMsg.st
```iecst
ACTION Act_OptP0600RcyMsg:

	//Recovery Message
	FOR i := 1 TO c_uiP0600TableSize DO

		IF tyP0600Alm.tyAlm.a_tyHotspotAlm[i].bRtCompl = TRUE THEN
			tyP0600Alm.tyAlm.a_tyHotspotAlm[i].bRtCompl	:= FALSE;

			tyP0600Alm.tyRcyMsg.tyTxtMsg.udiValueIdx := p_tyAlarmRcyList[i];

			IF tyP0600Alm.tyRcyMsg.tyTxtMsg.udiValueIdx <> 0 AND tyP0600Alm.tyAlm.tyBtnHistory.bValue = FALSE THEN
				p_tyC0010RcyMsg ACCESS ADR(tyP0600Alm.tyRcyMsg);
			ELSE
				p_tyC0010RcyMsg ACCESS ADR(tyP0600Alm.tyRcyMsgHide);
			END_IF

		END_IF

	END_FOR

	// Close Recovery Message
	IF tyP0600Alm.tyRcyMsg.tyHotspotClose.bRtCompl THEN
		tyP0600Alm.tyRcyMsg.tyHotspotClose.bRtCompl := FALSE;

		p_tyC0010RcyMsg ACCESS ADR(tyP0600Alm.tyRcyMsgHide);
	END_IF

END_ACTION
```

#### Act_EntP0700Disp.st
```iecst
ACTION Act_EntP0700Disp:

	//Access Address
	p_tyC0005Main ACCESS ADR(tyCommon.tyMain);

	p_tyC0007Notif ACCESS ADR(tyCommon.tyNotif);

	p_tyC0008MsgBox ACCESS ADR(tyP0700LFCtrl.tyMsgBoxHide);

	p_tyC0009Info ACCESS ADR(tyCommon.tyInfo);

	p_tyC0011Loading ACCESS ADR(tyCommon.tyLoading);

	p_tyP0700LFCtrl ACCESS ADR(tyP0700LFCtrl.tyLdr);

	//Run
	bLeaderRun	:= TRUE;

END_ACTION
```

#### Act_ExitP0700.st
```iecst
ACTION Act_ExitP0700:

	IF NOT(tyP0700LFCtrl.tyLdr.tyBtnChgAll.bRtCompl OR tyP0700LFCtrl.tyLdr.tyBtnChgSeqAuto.bRtCompl OR tyP0700LFCtrl.tyLdr.tyBtnChgSeqMnl.bRtCompl OR tyP0700LFCtrl.tyLdr.tyBtnSyncTm.bRtCompl) THEN
		bLeaderRun	:= FALSE;
		bLFRunInBG	:= FALSE;
	ELSE
		bLFRunInBG	:= TRUE;
	END_IF

	usiChgPage	:= 1;

END_ACTION
```

#### Act_OptP0700LFLeaderCtrl.st
```iecst
ACTION Act_OptP0700LFLeaderCtrl:

	CASE usiLFLeaderCtrlStep OF
		0:	//Confirmation Message - Execute Ask
			IF tyP0700LFCtrl.tyLdr.tyBtnChgAll.bRtCompl THEN

				p_tyC0008MsgBox ACCESS ADR(tyP0700LFCtrl.tyMsgBoxChgAllAsk);

				IF tyP0700LFCtrl.tyMsgBoxChgAllAsk.tyBtnYes.bRtCompl = TRUE THEN
					tyP0700LFCtrl.tyMsgBoxChgAllAsk.tyBtnYes.bRtCompl	:= FALSE;
					tyP0700LFCtrl.tyMsgBoxChgAllAsk.tyBtnYes.bValue		:= FALSE;

					p_tyC0008MsgBox ACCESS ADR(tyP0700LFCtrl.tyMsgBoxHide);

					tyP0700LFCtrl.tyLdr.tyBtnChgAll.bValue		:= TRUE;

					usiLFLeaderCtrlStep	:= 2;

				ELSIF tyP0700LFCtrl.tyMsgBoxChgAllAsk.tyBtnNo.bRtCompl = TRUE THEN
					tyP0700LFCtrl.tyMsgBoxChgAllAsk.tyBtnNo.bRtCompl	:= FALSE;
					tyP0700LFCtrl.tyMsgBoxChgAllAsk.tyBtnNo.bValue		:= FALSE;

					p_tyC0008MsgBox ACCESS ADR(tyP0700LFCtrl.tyMsgBoxHide);

					tyP0700LFCtrl.tyLdr.tyBtnChgAll.bValue		:= FALSE;
					tyP0700LFCtrl.tyLdr.tyBtnChgAll.bRtCompl	:= FALSE;

				END_IF

			ELSIF tyP0700LFCtrl.tyLdr.tyBtnChgSeqAuto.bRtCompl THEN

				p_tyC0008MsgBox ACCESS ADR(tyP0700LFCtrl.tyMsgBoxChgSeqAutoAsk);

				IF tyP0700LFCtrl.tyMsgBoxChgSeqAutoAsk.tyBtnYes.bRtCompl = TRUE THEN
					tyP0700LFCtrl.tyMsgBoxChgSeqAutoAsk.tyBtnYes.bRtCompl	:= FALSE;
					tyP0700LFCtrl.tyMsgBoxChgSeqAutoAsk.tyBtnYes.bValue		:= FALSE;

					p_tyC0008MsgBox ACCESS ADR(tyP0700LFCtrl.tyMsgBoxHide);

					tyP0700LFCtrl.tyLdr.tyBtnChgSeqAuto.bValue		:= TRUE;

					usiLFLeaderCtrlStep	:= 2;

				ELSIF tyP0700LFCtrl.tyMsgBoxChgSeqAutoAsk.tyBtnNo.bRtCompl = TRUE THEN
					tyP0700LFCtrl.tyMsgBoxChgSeqAutoAsk.tyBtnNo.bRtCompl	:= FALSE;
					tyP0700LFCtrl.tyMsgBoxChgSeqAutoAsk.tyBtnNo.bValue		:= FALSE;

					p_tyC0008MsgBox ACCESS ADR(tyP0700LFCtrl.tyMsgBoxHide);

					tyP0700LFCtrl.tyLdr.tyBtnChgSeqAuto.bValue		:= FALSE;
					tyP0700LFCtrl.tyLdr.tyBtnChgSeqAuto.bRtCompl	:= FALSE;

				END_IF

			ELSIF tyP0700LFCtrl.tyLdr.tyBtnChgSeqMnl.bRtCompl THEN

				p_tyC0008MsgBox ACCESS ADR(tyP0700LFCtrl.tyMsgBoxChgSeqMnlAsk);

				IF tyP0700LFCtrl.tyMsgBoxChgSeqMnlAsk.tyBtnYes.bRtCompl = TRUE THEN
					tyP0700LFCtrl.tyMsgBoxChgSeqMnlAsk.tyBtnYes.bRtCompl	:= FALSE;
					tyP0700LFCtrl.tyMsgBoxChgSeqMnlAsk.tyBtnYes.bValue		:= FALSE;

					p_tyC0008MsgBox ACCESS ADR(tyP0700LFCtrl.tyMsgBoxHide);

					tyP0700LFCtrl.tyLdr.tyBtnChgSeqMnl.bValue	:= TRUE;

					usiLFLeaderCtrlStep	:= 2;

				ELSIF tyP0700LFCtrl.tyMsgBoxChgSeqMnlAsk.tyBtnNo.bRtCompl = TRUE THEN
					tyP0700LFCtrl.tyMsgBoxChgSeqMnlAsk.tyBtnNo.bRtCompl		:= FALSE;
					tyP0700LFCtrl.tyMsgBoxChgSeqMnlAsk.tyBtnNo.bValue		:= FALSE;

					p_tyC0008MsgBox ACCESS ADR(tyP0700LFCtrl.tyMsgBoxHide);

					tyP0700LFCtrl.tyLdr.tyBtnChgSeqMnl.bValue	:= FALSE;
					tyP0700LFCtrl.tyLdr.tyBtnChgSeqMnl.bRtCompl	:= FALSE;

				END_IF

			ELSIF tyP0700LFCtrl.tyLdr.tyBtnSyncTm.bRtCompl THEN

				p_tyC0008MsgBox ACCESS ADR(tyP0700LFCtrl.tyMsgBoxSyncPLCTmAsk);

				IF tyP0700LFCtrl.tyMsgBoxSyncPLCTmAsk.tyBtnYes.bRtCompl = TRUE THEN
					tyP0700LFCtrl.tyMsgBoxSyncPLCTmAsk.tyBtnYes.bRtCompl	:= FALSE;
					tyP0700LFCtrl.tyMsgBoxSyncPLCTmAsk.tyBtnYes.bValue		:= FALSE;

					p_tyC0008MsgBox ACCESS ADR(tyP0700LFCtrl.tyMsgBoxHide);

					tyP0700LFCtrl.tyLdr.tyBtnSyncTm.bValue		:= TRUE;

					usiLFLeaderCtrlStep	:= 2;

				ELSIF tyP0700LFCtrl.tyMsgBoxSyncPLCTmAsk.tyBtnNo.bRtCompl = TRUE THEN
					tyP0700LFCtrl.tyMsgBoxSyncPLCTmAsk.tyBtnNo.bRtCompl		:= FALSE;
					tyP0700LFCtrl.tyMsgBoxSyncPLCTmAsk.tyBtnNo.bValue		:= FALSE;

					p_tyC0008MsgBox ACCESS ADR(tyP0700LFCtrl.tyMsgBoxHide);

					tyP0700LFCtrl.tyLdr.tyBtnSyncTm.bValue		:= FALSE;
					tyP0700LFCtrl.tyLdr.tyBtnSyncTm.bRtCompl	:= FALSE;

				END_IF

			END_IF

		1:	//Confirmation Message - Terminate Ask
			p_tyC0008MsgBox ACCESS ADR(tyP0700LFCtrl.tyMsgBoxTerminateOpsAsk);

			IF tyP0700LFCtrl.tyMsgBoxTerminateOpsAsk.tyBtnYes.bRtCompl = TRUE THEN
				tyP0700LFCtrl.tyMsgBoxTerminateOpsAsk.tyBtnYes.bRtCompl	:= FALSE;
				tyP0700LFCtrl.tyMsgBoxTerminateOpsAsk.tyBtnYes.bValue	:= FALSE;

				p_tyC0008MsgBox ACCESS ADR(tyP0700LFCtrl.tyMsgBoxHide);

				usiLFLeaderCtrlStep	:= 3;

			ELSIF tyP0700LFCtrl.tyMsgBoxTerminateOpsAsk.tyBtnNo.bRtCompl = TRUE THEN
				tyP0700LFCtrl.tyMsgBoxTerminateOpsAsk.tyBtnNo.bRtCompl	:= FALSE;
				tyP0700LFCtrl.tyMsgBoxTerminateOpsAsk.tyBtnNo.bValue	:= FALSE;

				p_tyC0008MsgBox ACCESS ADR(tyP0700LFCtrl.tyMsgBoxHide);

				tyP0700LFCtrl.tyLdr.tyBtnChgAll.bValue		:= tyP0700LFCtrl.tyLdr.tyBtnChgAll.bRtCompl;
				tyP0700LFCtrl.tyLdr.tyBtnChgSeqAuto.bValue	:= tyP0700LFCtrl.tyLdr.tyBtnChgSeqAuto.bRtCompl;
				tyP0700LFCtrl.tyLdr.tyBtnChgSeqMnl.bValue	:= tyP0700LFCtrl.tyLdr.tyBtnChgSeqMnl.bRtCompl;
				tyP0700LFCtrl.tyLdr.tyBtnSyncTm.bValue		:= tyP0700LFCtrl.tyLdr.tyBtnSyncTm.bRtCompl;

				usiLFLeaderCtrlStep	:= 2;

			END_IF

			//Display
			tyP0700LFCtrl.tyLdr.tyBitmapChgAll.usiValueIdx		:= BOOL_TO_USINT(tyP0700LFCtrl.tyLdr.tyBtnChgAll.bRtCompl);
			tyP0700LFCtrl.tyLdr.tyBitmapChgSeqAuto.usiValueIdx	:= BOOL_TO_USINT(tyP0700LFCtrl.tyLdr.tyBtnChgSeqAuto.bRtCompl);
			tyP0700LFCtrl.tyLdr.tyBitmapChgSeqMnl.usiValueIdx	:= BOOL_TO_USINT(tyP0700LFCtrl.tyLdr.tyBtnChgSeqMnl.bRtCompl);
			tyP0700LFCtrl.tyLdr.tyBitmapSyncTm.usiValueIdx		:= BOOL_TO_USINT(tyP0700LFCtrl.tyLdr.tyBtnSyncTm.bRtCompl);

		2:	//Processing
			IF tyP0700LFCtrl.tyLdr.tyBtnChgAll.bRtCompl THEN
				eLFLeaderAct	:= LFActChgAllAuto;

				IF p_eLFLeaderStat = LFActChgAllAuto AND (p_eLFLeaderStatus = Done OR p_eLFLeaderStatus = Error) THEN
					usiLFLeaderCtrlStep	:= 3;
				ELSIF tyP0700LFCtrl.tyLdr.tyBtnChgAll.bValue = FALSE THEN
					usiLFLeaderCtrlStep	:= 1;
				END_IF

			ELSIF tyP0700LFCtrl.tyLdr.tyBtnChgSeqAuto.bRtCompl THEN
				eLFLeaderAct	:= LFActChgSeqAuto;

				IF p_eLFLeaderStat = LFActChgSeqAuto AND (p_eLFLeaderStatus = Done OR p_eLFLeaderStatus = Error) THEN
					usiLFLeaderCtrlStep	:= 3;
				ELSIF tyP0700LFCtrl.tyLdr.tyBtnChgSeqAuto.bValue = FALSE THEN
					usiLFLeaderCtrlStep	:= 1;
				END_IF

			ELSIF tyP0700LFCtrl.tyLdr.tyBtnChgSeqMnl.bRtCompl THEN
				eLFLeaderAct	:= LFActChgSeqMnl;

				IF p_eLFLeaderStat = LFActChgSeqMnl AND (p_eLFLeaderStatus = Done OR p_eLFLeaderStatus = Error) THEN
					usiLFLeaderCtrlStep	:= 3;
				ELSIF tyP0700LFCtrl.tyLdr.tyBtnChgSeqMnl.bValue = FALSE THEN
					usiLFLeaderCtrlStep	:= 1;
				END_IF

			ELSIF tyP0700LFCtrl.tyLdr.tyBtnSyncTm.bRtCompl THEN
				eLFLeaderAct	:= LFActSyncPLCTm;

				IF p_eLFLeaderStat = LFActSyncPLCTm AND (p_eLFLeaderStatus = Done OR p_eLFLeaderStatus = Error) THEN
					usiLFLeaderCtrlStep	:= 3;
				ELSIF tyP0700LFCtrl.tyLdr.tyBtnSyncTm.bValue = FALSE THEN
					usiLFLeaderCtrlStep	:= 1;
				END_IF

			END_IF

			//Display
			fbLFLeaderCtrlBlinkTm(IN := TRUE);
			IF fbLFLeaderCtrlBlinkTm.Q = TRUE THEN
				fbLFLeaderCtrlBlinkTm(IN := FALSE);

				tyP0700LFCtrl.tyLdr.tyBitmapChgAll.usiValueIdx		:= BOOL_TO_USINT(USINT_TO_BOOL(tyP0700LFCtrl.tyLdr.tyBitmapChgAll.usiValueIdx) XOR tyP0700LFCtrl.tyLdr.tyBtnChgAll.bRtCompl);
				tyP0700LFCtrl.tyLdr.tyBitmapChgSeqAuto.usiValueIdx	:= BOOL_TO_USINT(USINT_TO_BOOL(tyP0700LFCtrl.tyLdr.tyBitmapChgSeqAuto.usiValueIdx) XOR tyP0700LFCtrl.tyLdr.tyBtnChgSeqAuto.bRtCompl);
				tyP0700LFCtrl.tyLdr.tyBitmapChgSeqMnl.usiValueIdx	:= BOOL_TO_USINT(USINT_TO_BOOL(tyP0700LFCtrl.tyLdr.tyBitmapChgSeqMnl.usiValueIdx) XOR tyP0700LFCtrl.tyLdr.tyBtnChgSeqMnl.bRtCompl);
				tyP0700LFCtrl.tyLdr.tyBitmapSyncTm.usiValueIdx		:= BOOL_TO_USINT(USINT_TO_BOOL(tyP0700LFCtrl.tyLdr.tyBitmapSyncTm.usiValueIdx) XOR tyP0700LFCtrl.tyLdr.tyBtnSyncTm.bRtCompl);
			END_IF

		3:	//Complete Reset
			usiLFLeaderCtrlStep	:= 0;

			eLFLeaderAct	:= LFActIdle;

			fbLFLeaderCtrlBlinkTm(IN := FALSE);

			tyP0700LFCtrl.tyLdr.tyBitmapChgAll.usiValueIdx		:= 0;
			tyP0700LFCtrl.tyLdr.tyBitmapChgSeqAuto.usiValueIdx	:= 0;
			tyP0700LFCtrl.tyLdr.tyBitmapChgSeqMnl.usiValueIdx	:= 0;
			tyP0700LFCtrl.tyLdr.tyBitmapSyncTm.usiValueIdx		:= 0;

			tyP0700LFCtrl.tyLdr.tyBtnChgAll.bRtCompl			:= FALSE;
			tyP0700LFCtrl.tyLdr.tyBtnChgSeqAuto.bRtCompl		:= FALSE;
			tyP0700LFCtrl.tyLdr.tyBtnChgSeqMnl.bRtCompl			:= FALSE;
			tyP0700LFCtrl.tyLdr.tyBtnSyncTm.bRtCompl			:= FALSE;

			tyP0700LFCtrl.tyLdr.tyBtnChgAll.bValue				:= FALSE;
			tyP0700LFCtrl.tyLdr.tyBtnChgSeqAuto.bValue			:= FALSE;
			tyP0700LFCtrl.tyLdr.tyBtnChgSeqMnl.bValue			:= FALSE;
			tyP0700LFCtrl.tyLdr.tyBtnSyncTm.bValue				:= FALSE;

		4:
			p_tyC0008MsgBox ACCESS ADR(tyP0700LFCtrl.tyMsgBoxErrorAsk);

			IF tyP0700LFCtrl.tyMsgBoxErrorAsk.tyBtnNo.bRtCompl = TRUE THEN
				tyP0700LFCtrl.tyMsgBoxErrorAsk.tyBtnNo.bRtCompl	:= FALSE;
				tyP0700LFCtrl.tyMsgBoxErrorAsk.tyBtnNo.bValue	:= FALSE;

				p_tyC0008MsgBox ACCESS ADR(tyP0700LFCtrl.tyMsgBoxHide);

				usiLFLeaderCtrlStep	:= 3;

			END_IF

	END_CASE

END_ACTION
```

#### Act_OptP0700Mask.st
```iecst
ACTION Act_OptP0700Mask:

	//Mask
	IF p_eLFLeaderStatus = Error THEN
		fUIInRtStatOff(ADR(tyP0700LFCtrl.tyLdr.tyBtnChgAll.uiMaskRtStat));
		fUIInRtStatOff(ADR(tyP0700LFCtrl.tyLdr.tyBtnChgSeqAuto.uiMaskRtStat));
		fUIInRtStatOff(ADR(tyP0700LFCtrl.tyLdr.tyBtnChgSeqMnl.uiMaskRtStat));
		fUIInRtStatOff(ADR(tyP0700LFCtrl.tyLdr.tyBtnSyncTm.uiMaskRtStat));

	ELSIF tyP0700LFCtrl.tyLdr.tyBtnChgAll.bRtCompl THEN
		fUIInRtStatHide(ADR(tyP0700LFCtrl.tyLdr.tyBtnChgAll.uiMaskRtStat));
		fUIInRtStatOff(ADR(tyP0700LFCtrl.tyLdr.tyBtnChgSeqAuto.uiMaskRtStat));
		fUIInRtStatOff(ADR(tyP0700LFCtrl.tyLdr.tyBtnChgSeqMnl.uiMaskRtStat));
		fUIInRtStatOff(ADR(tyP0700LFCtrl.tyLdr.tyBtnSyncTm.uiMaskRtStat));

	ELSIF tyP0700LFCtrl.tyLdr.tyBtnChgSeqAuto.bRtCompl THEN
		fUIInRtStatOff(ADR(tyP0700LFCtrl.tyLdr.tyBtnChgAll.uiMaskRtStat));
		fUIInRtStatHide(ADR(tyP0700LFCtrl.tyLdr.tyBtnChgSeqAuto.uiMaskRtStat));
		fUIInRtStatOff(ADR(tyP0700LFCtrl.tyLdr.tyBtnChgSeqMnl.uiMaskRtStat));
		fUIInRtStatOff(ADR(tyP0700LFCtrl.tyLdr.tyBtnSyncTm.uiMaskRtStat));

	ELSIF tyP0700LFCtrl.tyLdr.tyBtnChgSeqMnl.bRtCompl THEN
		fUIInRtStatOff(ADR(tyP0700LFCtrl.tyLdr.tyBtnChgAll.uiMaskRtStat));
		fUIInRtStatOff(ADR(tyP0700LFCtrl.tyLdr.tyBtnChgSeqAuto.uiMaskRtStat));
		fUIInRtStatHide(ADR(tyP0700LFCtrl.tyLdr.tyBtnChgSeqMnl.uiMaskRtStat));
		fUIInRtStatOff(ADR(tyP0700LFCtrl.tyLdr.tyBtnSyncTm.uiMaskRtStat));

	ELSIF tyP0700LFCtrl.tyLdr.tyBtnSyncTm.bRtCompl THEN
		fUIInRtStatOff(ADR(tyP0700LFCtrl.tyLdr.tyBtnChgAll.uiMaskRtStat));
		fUIInRtStatOff(ADR(tyP0700LFCtrl.tyLdr.tyBtnChgSeqAuto.uiMaskRtStat));
		fUIInRtStatOff(ADR(tyP0700LFCtrl.tyLdr.tyBtnChgSeqMnl.uiMaskRtStat));
		fUIInRtStatHide(ADR(tyP0700LFCtrl.tyLdr.tyBtnSyncTm.uiMaskRtStat));

	ELSE
		fUIInRtStatHide(ADR(tyP0700LFCtrl.tyLdr.tyBtnChgAll.uiMaskRtStat));
		fUIInRtStatHide(ADR(tyP0700LFCtrl.tyLdr.tyBtnChgSeqAuto.uiMaskRtStat));
		fUIInRtStatHide(ADR(tyP0700LFCtrl.tyLdr.tyBtnChgSeqMnl.uiMaskRtStat));
		fUIInRtStatHide(ADR(tyP0700LFCtrl.tyLdr.tyBtnSyncTm.uiMaskRtStat));

	END_IF

END_ACTION
```

#### Act_OptP0700Table.st
```iecst
ACTION Act_OptP0700Table:

	//Call Table FB
	fbP0700Table.sVisuNm			:= tyP0700Table.sVisuNm;
	fbP0700Table.udiWorkAreaStartX	:= 14;
	fbP0700Table.udiWorkAreaEndX	:= 475;
	fbP0700Table.udiWorkAreaStartY	:= 45;
	fbP0700Table.udiWorkAreaEndY	:= 217;
	fbP0700Table.udiMinXDist		:= 20;
	fbP0700Table.udiMinYDist		:= 20;
	fbP0700Table.uiSlideScale		:= c_uiP0700TableSize;
	fbP0700Table.iTotalData			:= UDINT_TO_INT(c_diLFClntNum);
	fbP0700Table.iTotalRow			:= c_uiP0700TableSize;
	fbP0700Table(uiSliderStatus 	:= tyP0700LFCtrl.tyLdr.tyTable1List.tyUISlider.uiRtStat , a_tyUIHotspot := tyP0700LFCtrl.tyLdr.tyTable1List.a_tyHotspot , uiTablePos := tyP0700Table.uiTablePos , iSliderPos := tyP0700LFCtrl.tyLdr.tyTable1List.tyUISlider.iValue);

	tyP0700Table.uiSelectedRow		:= fbP0700Table.uiSelectedRow;
	tyP0700Table.bTableActive		:= fbP0700Table.bTableActive;
	tyP0700Table.bSliderActive		:= fbP0700Table.bSliderActive;

	//Table Content
	IF tyP0700Table.bTableActive = TRUE OR tyP0700Table.bSliderActive = TRUE THEN
		FOR i := 1 TO c_uiP0700TableSize DO
			tyP0700LFCtrl.tyLdr.tyTable1List.a_tyStringDataCol0[i].sValue	:= UINT_TO_STRING(tyP0700Table.uiTablePos + i - 1);
		END_FOR
	END_IF

	//Update Status & Current Recipe
	FOR i := 1 TO c_uiP0700TableSize DO
		tyP0700LFCtrl.tyLdr.tyTable1List.a_tyStringDataCol1[i].sValue	:= p_tyLFLeaderFollowerToLeaderTag[tyP0700Table.uiTablePos + i - 1].sMcNm;
		tyP0700LFCtrl.tyLdr.tyTable1List.a_tyStringDataCol2[i].sValue	:= p_tyMcParamCurr.a_sLFIPAddr[tyP0700Table.uiTablePos + i - 1];
		tyP0700LFCtrl.tyLdr.tyTable1List.a_tyStringDataCol4[i].sValue	:= p_tyLFLeaderFollowerToLeaderTag[tyP0700Table.uiTablePos + i - 1].sCurrProdRcp;

		IF p_tyMcParamCurr.a_sLFIPAddr[tyP0700Table.uiTablePos + i - 1] = '' THEN
			tyP0700LFCtrl.tyLdr.tyTable1List.a_tyTxtDataCol3[i].usiValueIdx	:= 0;	//Empty
		ELSIF p_tyMcParamCurr.a_sLFIPAddr[tyP0700Table.uiTablePos + i - 1] = '0000' THEN
			tyP0700LFCtrl.tyLdr.tyTable1List.a_tyTxtDataCol3[i].usiValueIdx	:= 3;	//Third Party
		ELSIF p_tyMcParamCurr.a_bLFOnline[tyP0700Table.uiTablePos + i - 1] = FALSE THEN
			tyP0700LFCtrl.tyLdr.tyTable1List.a_tyTxtDataCol3[i].usiValueIdx	:= 9;	//Offline
		ELSIF p_tyMcParamCurr.a_sLFIPAddr[tyP0700Table.uiTablePos + i - 1] = p_sHWInfoIPAddr THEN
			tyP0700LFCtrl.tyLdr.tyTable1List.a_tyTxtDataCol3[i].usiValueIdx	:= 4;	//Leader
		ELSIF p_tyLFLeaderFollowerToLeaderTag[tyP0700Table.uiTablePos + i - 1].bSectionLeader = TRUE THEN
			tyP0700LFCtrl.tyLdr.tyTable1List.a_tyTxtDataCol3[i].usiValueIdx	:= 5;	//Section Leader
		ELSIF p_tyLFLeaderFollowerInfo[tyP0700Table.uiTablePos + i - 1].bOnline = FALSE THEN
			tyP0700LFCtrl.tyLdr.tyTable1List.a_tyTxtDataCol3[i].usiValueIdx	:= 9;	//Offline
		ELSE
			IF p_tyLFLeaderFollowerToLeaderTag[tyP0700Table.uiTablePos + i - 1].eCurrMachineStat=Run THEN
				IF p_tyLFLeaderFollowerToLeaderTag[tyP0700Table.uiTablePos + i - 1].eCurrMachineStat=Warning THEN
					tyP0700LFCtrl.tyLdr.tyTable1List.a_tyTxtDataCol3[i].usiValueIdx	:= 2;	//Warning
				ELSE
					tyP0700LFCtrl.tyLdr.tyTable1List.a_tyTxtDataCol3[i].usiValueIdx	:= 6;	//Run
				END_IF
			ELSE
				IF p_tyLFLeaderFollowerToLeaderTag[tyP0700Table.uiTablePos + i - 1].eCurrMachineStat=InError THEN
					tyP0700LFCtrl.tyLdr.tyTable1List.a_tyTxtDataCol3[i].usiValueIdx	:= 1;	//Error
				ELSIF p_tyLFLeaderFollowerToLeaderTag[tyP0700Table.uiTablePos + i - 1].eCurrMachineStat=Warning THEN
					tyP0700LFCtrl.tyLdr.tyTable1List.a_tyTxtDataCol3[i].usiValueIdx	:= 2;	//Warning
				ELSIF p_tyLFLeaderFollowerToLeaderTag[tyP0700Table.uiTablePos + i - 1].eCurrMachineStat=Manual THEN
					tyP0700LFCtrl.tyLdr.tyTable1List.a_tyTxtDataCol3[i].usiValueIdx	:= 8;	//Manual
				ELSE
					tyP0700LFCtrl.tyLdr.tyTable1List.a_tyTxtDataCol3[i].usiValueIdx	:= 7;	//Stop
				END_IF
			END_IF
		END_IF
	END_FOR

	//Update Color
	FOR i := 1 TO c_uiP0700TableSize DO

		IF p_tyMcParamCurr.a_sLFIPAddr[tyP0700Table.uiTablePos + i - 1] = '' THEN
			tyP0700LFCtrl.tyLdr.tyTable1List.a_tyTxtDataCol3[i].usiColor	:= 0;	//Empty
		ELSIF p_tyMcParamCurr.a_sLFIPAddr[tyP0700Table.uiTablePos + i - 1] = '0000' THEN
			tyP0700LFCtrl.tyLdr.tyTable1List.a_tyTxtDataCol3[i].usiColor	:= 0;	//Third Party
		ELSIF p_tyMcParamCurr.a_bLFOnline[tyP0700Table.uiTablePos + i - 1] = FALSE THEN
			tyP0700LFCtrl.tyLdr.tyTable1List.a_tyTxtDataCol3[i].usiColor	:= 3;	//Offline
		ELSIF p_tyMcParamCurr.a_sLFIPAddr[tyP0700Table.uiTablePos + i - 1] = p_sHWInfoIPAddr THEN
			IF p_bOpsRun THEN
				tyP0700LFCtrl.tyLdr.tyTable1List.a_tyTxtDataCol3[i].usiColor	:= 1;	//Leader Run
			ELSE
				tyP0700LFCtrl.tyLdr.tyTable1List.a_tyTxtDataCol3[i].usiColor	:= 2;	//Leader Stop
			END_IF
		ELSIF p_tyLFLeaderFollowerToLeaderTag[tyP0700Table.uiTablePos + i - 1].bSectionLeader = TRUE THEN
			IF p_tyLFLeaderFollowerToLeaderTag[tyP0700Table.uiTablePos + i - 1].eCurrMachineStat=Run THEN
				tyP0700LFCtrl.tyLdr.tyTable1List.a_tyTxtDataCol3[i].usiColor	:= 1;	//Section Leader Run
			ELSE
				tyP0700LFCtrl.tyLdr.tyTable1List.a_tyTxtDataCol3[i].usiColor	:= 2;	//Section Leader Stop
			END_IF
		ELSIF p_tyLFLeaderFollowerInfo[tyP0700Table.uiTablePos + i - 1].bOnline = FALSE THEN
			tyP0700LFCtrl.tyLdr.tyTable1List.a_tyTxtDataCol3[i].usiColor	:= 3;	//Offline
		ELSE
			IF p_tyLFLeaderFollowerToLeaderTag[tyP0700Table.uiTablePos + i - 1].eCurrMachineStat=Run THEN
				IF p_tyLFLeaderFollowerToLeaderTag[tyP0700Table.uiTablePos + i - 1].eCurrMachineStat=Warning THEN
					tyP0700LFCtrl.tyLdr.tyTable1List.a_tyTxtDataCol3[i].usiColor	:= 4;	//Warning
				ELSE
					tyP0700LFCtrl.tyLdr.tyTable1List.a_tyTxtDataCol3[i].usiColor	:= 1;	//Run
				END_IF
			ELSE
				IF p_tyLFLeaderFollowerToLeaderTag[tyP0700Table.uiTablePos + i - 1].eCurrMachineStat=InError THEN
					tyP0700LFCtrl.tyLdr.tyTable1List.a_tyTxtDataCol3[i].usiColor	:= 2;	//Error
				ELSIF p_tyLFLeaderFollowerToLeaderTag[tyP0700Table.uiTablePos + i - 1].eCurrMachineStat=Warning THEN
					tyP0700LFCtrl.tyLdr.tyTable1List.a_tyTxtDataCol3[i].usiColor	:= 4;	//Warning
				ELSIF p_tyLFLeaderFollowerToLeaderTag[tyP0700Table.uiTablePos + i - 1].eCurrMachineStat=Manual THEN
					tyP0700LFCtrl.tyLdr.tyTable1List.a_tyTxtDataCol3[i].usiColor	:= 6;	//Manual
				ELSE
					tyP0700LFCtrl.tyLdr.tyTable1List.a_tyTxtDataCol3[i].usiColor	:= 5;	//Stop
				END_IF
			END_IF
		END_IF

	END_FOR

END_ACTION
```

#### Act_EntP0900Disp.st
```iecst
ACTION Act_EntP0900Disp:

	//Access Address
	p_tyC0005Main ACCESS ADR(tyCommon.tyMain);

	p_tyC0007Notif ACCESS ADR(tyCommon.tyNotif);

	p_tyC0008MsgBox ACCESS ADR(tyP0900GenIn.tyMsgBoxHide);

	p_tyC0009Info ACCESS ADR(tyCommon.tyInfo);

	p_tyC0011Loading ACCESS ADR(tyCommon.tyLoading);

	p_tyP0900GenIn ACCESS ADR(tyP0900GenIn.tyGenIn);

END_ACTION
```

#### Act_OptP0900ReadDI.st
```iecst
ACTION Act_OptP0900ReadDI:

	tyP0900GenIn.tyGenIn.tyBtnSafety.bValue		:= p_tyDI.bSafetyRlySig;
	tyP0900GenIn.tyGenIn.tyBtnEStop.bValue		:= p_tyDI.bEStopSig;
	tyP0900GenIn.tyGenIn.tyBtnCoverSW.bValue	:= p_tyDI.bCoverSWSig;

	tyP0900GenIn.tyGenIn.tyBtnThermalPrtSig.bValue	:= p_tyDI.bThermalPrtSig;
	tyP0900GenIn.tyGenIn.tyBtnUSWidthChkSen.bValue	:= p_tyDI.bUSWidthChkSen;
	tyP0900GenIn.tyGenIn.tyBtnDSWidthChkSen.bValue	:= p_tyDI.bDSWidthChkSen;

	// ADD
	tyP0900GenIn.tyGenIn.tyBtnSafetySigFromDS.bValue  := p_tyDI.bSafetySigFromDS;
	tyP0900GenIn.tyGenIn.tyBtnSafetySigFromUS.bValue  := p_tyDI.bSafetySigFromUS;
	tyP0900GenIn.tyGenIn.tyBtnUlkCoverFromDS.bValue   := p_tyDI.bUnlockCoverSigFromDS;
	tyP0900GenIn.tyGenIn.tyBtnUlkCoverFromUS.bValue   := p_tyDI.bUnlockCoverSigFromUS;
	tyP0900GenIn.tyGenIn.tyBtnUnlkCovPB.bValue        := p_tyDI.bCoverUnlockPB1;
	tyP0900GenIn.tyGenIn.tyBtnTopCovSwSIg.bValue      :=  p_tyDI.bCoverSWSig2;
END_ACTION
```

#### Act_EntP0910Disp.st
```iecst
ACTION Act_EntP0910Disp:

	//Access Address
	p_tyC0005Main ACCESS ADR(tyCommon.tyMain);

	p_tyC0007Notif ACCESS ADR(tyCommon.tyNotif);

	p_tyC0008MsgBox ACCESS ADR(tyP0910GenOut.tyMsgBoxHide);

	p_tyC0009Info ACCESS ADR(tyCommon.tyInfo);

	p_tyC0011Loading ACCESS ADR(tyCommon.tyLoading);

	p_tyP0910GenOut ACCESS ADR(tyP0910GenOut.tyGenOut);

END_ACTION
```

#### Act_OptP0910WriteDO.st
```iecst
ACTION Act_OptP0910WriteDO:

	//Safety Relay
	IF tyP0910GenOut.tyGenOut.tyBtnSafety.bRtCompl = TRUE THEN

		IF tyP0910GenOut.tyGenOut.tyBtnSafety.bValue = TRUE THEN
			eRstErrAct	:= RstErrActSetSafetyRlyRst;

			IF p_eRstErrStat = RstErrActSetSafetyRlyRst AND p_eRstErrStatus = Done THEN
				eRstErrAct	:= RstErrActIdle;

				tyP0910GenOut.tyGenOut.tyBtnSafety.bRtCompl	:= FALSE;
			END_IF

		ELSE
			eRstErrAct	:= RstErrActRstSafetyRlyRst;

			IF p_eRstErrStat = RstErrActRstSafetyRlyRst AND p_eRstErrStatus = Done THEN
				eRstErrAct	:= RstErrActIdle;

				tyP0910GenOut.tyGenOut.tyBtnSafety.bRtCompl	:= FALSE;
			END_IF

		END_IF

	END_IF

	// TL Green
	IF tyP0910GenOut.tyGenOut.tyBtnTLGreen.bRtCompl = TRUE THEN
		IF tyP0910GenOut.tyGenOut.tyBtnTLGreen.bValue = TRUE THEN
			eTLBuzAct	:= TLBuzActSetGreen;

			IF p_eTLBuzStat = TLBuzActSetGreen AND p_eTLBuzStatus = Done THEN
				eTLBuzAct	:= TLBuzActIdle;

				tyP0910GenOut.tyGenOut.tyBtnTLGreen.bRtCompl	:= FALSE;
			END_IF
		ELSE
			eTLBuzAct	:= TLBuzActRstGreen;

			IF p_eTLBuzStat = TLBuzActRstGreen AND p_eTLBuzStatus = Done THEN
				eTLBuzAct	:= TLBuzActIdle;

				tyP0910GenOut.tyGenOut.tyBtnTLGreen.bRtCompl	:= FALSE;
			END_IF

		END_IF
	END_IF

	//TL Amber
	IF tyP0910GenOut.tyGenOut.tyBtnTLAmber.bRtCompl = TRUE THEN
		IF tyP0910GenOut.tyGenOut.tyBtnTLAmber.bValue = TRUE THEN
			eTLBuzAct	:= TLBuzActSetAmber;

			IF p_eTLBuzStat = TLBuzActSetAmber AND p_eTLBuzStatus = Done THEN
				eTLBuzAct	:= TLBuzActIdle;

				tyP0910GenOut.tyGenOut.tyBtnTLAmber.bRtCompl	:= FALSE;
			END_IF
		ELSE
			eTLBuzAct	:= TLBuzActRstAmber;

			IF p_eTLBuzStat = TLBuzActRstAmber AND p_eTLBuzStatus = Done THEN
				eTLBuzAct	:= TLBuzActIdle;

				tyP0910GenOut.tyGenOut.tyBtnTLAmber.bRtCompl	:= FALSE;
			END_IF

		END_IF
	END_IF

	//TL Red
	IF tyP0910GenOut.tyGenOut.tyBtnTLRed.bRtCompl = TRUE THEN
		IF tyP0910GenOut.tyGenOut.tyBtnTLRed.bValue = TRUE THEN
			eTLBuzAct	:= TLBuzActSetRed;

			IF p_eTLBuzStat = TLBuzActSetRed AND p_eTLBuzStatus = Done THEN
				eTLBuzAct	:= TLBuzActIdle;

				tyP0910GenOut.tyGenOut.tyBtnTLRed.bRtCompl	:= FALSE;
			END_IF
		ELSE
			eTLBuzAct	:= TLBuzActRstRed;

			IF p_eTLBuzStat = TLBuzActRstRed AND p_eTLBuzStatus = Done THEN
				eTLBuzAct	:= TLBuzActIdle;

				tyP0910GenOut.tyGenOut.tyBtnTLRed.bRtCompl	:= FALSE;
			END_IF

		END_IF
	END_IF

	//TL Blue
	IF tyP0910GenOut.tyGenOut.tyBtnTLBlue.bRtCompl = TRUE THEN
		IF tyP0910GenOut.tyGenOut.tyBtnTLBlue.bValue = TRUE THEN
			eTLBuzAct	:= TLBuzActSetBlue;

			IF p_eTLBuzStat = TLBuzActSetBlue AND p_eTLBuzStatus = Done THEN
				eTLBuzAct	:= TLBuzActIdle;

				tyP0910GenOut.tyGenOut.tyBtnTLBlue.bRtCompl	:= FALSE;
			END_IF
		ELSE
			eTLBuzAct	:= TLBuzActRstBlue;

			IF p_eTLBuzStat = TLBuzActRstBlue AND p_eTLBuzStatus = Done THEN
				eTLBuzAct	:= TLBuzActIdle;

				tyP0910GenOut.tyGenOut.tyBtnTLBlue.bRtCompl	:= FALSE;
			END_IF

		END_IF
	END_IF

	//TL White
	IF tyP0910GenOut.tyGenOut.tyBtnTLWhite.bRtCompl = TRUE THEN
		IF tyP0910GenOut.tyGenOut.tyBtnTLWhite.bValue = TRUE THEN
			eTLBuzAct	:= TLBuzActSetWhite;

			IF p_eTLBuzStat = TLBuzActSetWhite AND p_eTLBuzStatus = Done THEN
				eTLBuzAct	:= TLBuzActIdle;

				tyP0910GenOut.tyGenOut.tyBtnTLWhite.bRtCompl	:= FALSE;
			END_IF
		ELSE
			eTLBuzAct	:= TLBuzActRstWhite;

			IF p_eTLBuzStat = TLBuzActRstWhite AND p_eTLBuzStatus = Done THEN
				eTLBuzAct	:= TLBuzActIdle;

				tyP0910GenOut.tyGenOut.tyBtnTLWhite.bRtCompl	:= FALSE;
			END_IF

		END_IF
	END_IF

	//TL Buzzer
	IF tyP0910GenOut.tyGenOut.tyBtnBuzzer.bRtCompl = TRUE THEN
		IF tyP0910GenOut.tyGenOut.tyBtnBuzzer.bValue = TRUE THEN
			eTLBuzAct	:= TLBuzActSetBuz;

			IF p_eTLBuzStat = TLBuzActSetBuz AND p_eTLBuzStatus = Done THEN
				eTLBuzAct	:= TLBuzActIdle;

				tyP0910GenOut.tyGenOut.tyBtnBuzzer.bRtCompl	:= FALSE;
			END_IF
		ELSE
			eTLBuzAct	:= TLBuzActRstBuz;

			IF p_eTLBuzStat = TLBuzActRstBuz AND p_eTLBuzStatus = Done THEN
				eTLBuzAct	:= TLBuzActIdle;

				tyP0910GenOut.tyGenOut.tyBtnBuzzer.bRtCompl	:= FALSE;
			END_IF

		END_IF
	END_IF

	// ADD
	// ADD

	//  Safety Sig to DS
	IF tyP0910GenOut.tyGenOut.tyBtnSftSigToUSDS.bRtCompl = TRUE THEN
		IF tyP0910GenOut.tyGenOut.tyBtnSftSigToUSDS.bValue = TRUE THEN
			bMnlModMachineSafetySigToDS		:= TRUE;
			tyP0910GenOut.tyGenOut.tyBtnSftSigToUSDS.bRtCompl		:= FALSE;
			//
		ELSE
			bMnlModMachineSafetySigToDS		:= FALSE;
			tyP0910GenOut.tyGenOut.tyBtnSftSigToUSDS.bRtCompl		:= FALSE;
			//
		END_IF
		//
	END_IF

	//  Top Cover Unlock Sig to DS
	IF 	tyP0910GenOut.tyGenOut.tyBtnTopCovUlkUSDS.bRtCompl = TRUE THEN
		IF 	tyP0910GenOut.tyGenOut.tyBtnTopCovUlkUSDS.bValue = TRUE THEN
			bMnlModUnlockCover1Req		:= TRUE;
			tyP0910GenOut.tyGenOut.tyBtnTopCovUlkUSDS.bRtCompl		:= FALSE;

		ELSE
			bMnlModUnlockCover1Req		:= FALSE;
			tyP0910GenOut.tyGenOut.tyBtnTopCovUlkUSDS.bRtCompl		:= FALSE;

		END_IF

	END_IF

	//  Unlock Cover PB led
	IF tyP0910GenOut.tyGenOut.tyBtnUlkCovPBLED.bRtCompl = TRUE THEN
		IF tyP0910GenOut.tyGenOut.tyBtnUlkCovPBLED.bValue = TRUE THEN
			bMnlModCoverPBLED1		:= TRUE;
			tyP0910GenOut.tyGenOut.tyBtnUlkCovPBLED.bRtCompl		:= FALSE;

		ELSE
			bMnlModCoverPBLED1		:= FALSE;
			tyP0910GenOut.tyGenOut.tyBtnUlkCovPBLED.bRtCompl		:= FALSE;

		END_IF

	END_IF

	//  ByPass Top Cover
	IF tyP0910GenOut.tyGenOut.tyBtnUlkCovHoldRely.bRtCompl = TRUE THEN
		IF tyP0910GenOut.tyGenOut.tyBtnUlkCovHoldRely.bValue = TRUE THEN
			bMnlModBypassTopCover1		:= TRUE;
			tyP0910GenOut.tyGenOut.tyBtnUlkCovHoldRely.bRtCompl		:= FALSE;

		ELSE
			bMnlModBypassTopCover1		:= FALSE;
			tyP0910GenOut.tyGenOut.tyBtnUlkCovHoldRely.bRtCompl		:= FALSE;

		END_IF

	END_IF

	//  Safety Top Cover Switch Coil
	IF tyP0910GenOut.tyGenOut.tyBtnSftUlkCovSWCoil.bRtCompl = TRUE THEN
		IF tyP0910GenOut.tyGenOut.tyBtnSftUlkCovSWCoil.bValue = TRUE THEN
			bMnlModTopCoverSwitch1		:= TRUE;
			tyP0910GenOut.tyGenOut.tyBtnSftUlkCovSWCoil.bRtCompl		:= FALSE;

		ELSE
			bMnlModTopCoverSwitch1		:= FALSE;
			tyP0910GenOut.tyGenOut.tyBtnSftUlkCovSWCoil.bRtCompl		:= FALSE;

		END_IF

	END_IF

END_ACTION
```

#### Act_OptP0910RstMnl.st
```iecst
ACTION Act_OptP0910RstMnl:

	IF EDGEPOS((bUIManualMod = FALSE) OR (p_eTLBuzStatus = Error) OR (p_eRstErrStatus = Error)) THEN

		eTLBuzAct	:= TLBuzActIdle;

		tyP0910GenOut.tyGenOut.tyBtnTLGreen.bValue	:= FALSE;
		tyP0910GenOut.tyGenOut.tyBtnTLAmber.bValue	:= FALSE;
		tyP0910GenOut.tyGenOut.tyBtnTLWhite.bValue	:= FALSE;
		tyP0910GenOut.tyGenOut.tyBtnTLRed.bValue	:= FALSE;
		tyP0910GenOut.tyGenOut.tyBtnBuzzer.bValue	:= FALSE;
		tyP0910GenOut.tyGenOut.tyBtnSafety.bValue	:= FALSE;

		// ADD
		tyP0910GenOut.tyGenOut.tyBtnSftSigToUSDS.bValue 	:= FALSE;
		tyP0910GenOut.tyGenOut.tyBtnSftUlkCovSWCoil.bValue	:= FALSE;
		tyP0910GenOut.tyGenOut.tyBtnTopCovUlkUSDS.bValue	:=FALSE;
		tyP0910GenOut.tyGenOut.tyBtnUlkCovPBLED.bValue		:= FALSE;
		tyP0910GenOut.tyGenOut.tyBtnUlkCovHoldRely.bValue	:= FALSE;
	END_IF

END_ACTION
```

#### Act_EntP0920Disp.st
```iecst
ACTION Act_EntP0920Disp:

	//Access Address
	p_tyC0002FullMask ACCESS ADR(tyP0920MtrNPneuCtrl.tyFullMaskHide);

	p_tyC0005Main ACCESS ADR(tyCommon.tyMain);

	p_tyC0007Notif ACCESS ADR(tyCommon.tyNotif);

	p_tyC0008MsgBox ACCESS ADR(tyP0920MtrNPneuCtrl.tyMsgBoxHide);

	p_tyC0009Info ACCESS ADR(tyCommon.tyInfo);

	p_tyC0011Loading ACCESS ADR(tyCommon.tyLoading);

	p_tyP0920MtrNPneuCtrl ACCESS ADR(tyP0920MtrNPneuCtrl.tyMtrNPneuCtrl);

	//AW Display
	tyP0920MtrNPneuCtrl.tyMtrNPneuCtrl.tyBtnAW.uiMaskRtStat.0		:= NOT(p_tyNtParamCurr.bAWPrep AND p_tyMcParamCurr.bAWDis);

	//Stopper Display
	tyP0920MtrNPneuCtrl.tyMtrNPneuCtrl.tyBtnStopper.uiMaskRtStat.0	:= NOT(p_tyNtParamCurr.bProjStopperPrep AND p_tyMcParamCurr.bStopperDis);

	//Clamp No RS Display
	tyP0920MtrNPneuCtrl.tyMtrNPneuCtrl.tyBtnClampNoRS.uiMaskRtStat.0	:= NOT(p_tyNtParamCurr.bProjClampPrep AND (p_tyNtParamCurr.eProjClampOption=ClampNoRS) AND p_tyMcParamCurr.bClampDis);

	//Clamp With RS Display
	tyP0920MtrNPneuCtrl.tyMtrNPneuCtrl.tyBtnClampWithRS.uiMaskRtStat.0	:= NOT(p_tyNtParamCurr.bProjClampPrep AND (p_tyNtParamCurr.eProjClampOption=ThreeClampsWithRS) AND p_tyMcParamCurr.bClampDis);

	//Shutter Display
	tyP0920MtrNPneuCtrl.tyMtrNPneuCtrl.tyBtnShutter.uiMaskRtStat.0		:= NOT((p_tyNtParamCurr.bProjInletShutPrep AND p_tyMcParamCurr.bInShutterDis) OR (p_tyNtParamCurr.bProjOutletShutPrep AND p_tyMcParamCurr.bOutShutterDis));

END_ACTION
```

#### Act_OptP0920FullMask.st
```iecst
ACTION Act_OptP0920FullMask:

	IF eCurrPage = UIP0920MtrNPneuCtrl THEN

		IF p_tyDI.bEStopSig = FALSE THEN
			p_tyC0002FullMask ACCESS ADR(tyP0920MtrNPneuCtrl.tyFullMaskEStop);

		ELSIF p_tyDI.bCoverSWSig = FALSE THEN
			p_tyC0002FullMask ACCESS ADR(tyP0920MtrNPneuCtrl.tyFullMaskCWSig);

		ELSIF p_tyDI.bSafetyRlySig = FALSE THEN
			p_tyC0002FullMask ACCESS ADR(tyP0920MtrNPneuCtrl.tyFullMaskSafetyRly);

		ELSE
			p_tyC0002FullMask ACCESS ADR(tyP0920MtrNPneuCtrl.tyFullMaskHide);

		END_IF

	END_IF

END_ACTION
```

#### Act_OptP0920ChgPage.st
```iecst
ACTION Act_OptP0920ChgPage:

	IF tyP0920MtrNPneuCtrl.tyMtrNPneuCtrl.tyBtnStopper.bRtCompl THEN
		tyP0920MtrNPneuCtrl.tyMtrNPneuCtrl.tyBtnStopper.bRtCompl	:= FALSE;
		tyP0920MtrNPneuCtrl.tyMtrNPneuCtrl.tyBtnStopper.bValue		:= FALSE;

		eChgPage			:= UIP0923Stopper;

	ELSIF tyP0920MtrNPneuCtrl.tyMtrNPneuCtrl.tyBtnConv.bRtCompl THEN
		tyP0920MtrNPneuCtrl.tyMtrNPneuCtrl.tyBtnConv.bRtCompl		:= FALSE;
		tyP0920MtrNPneuCtrl.tyMtrNPneuCtrl.tyBtnConv.bValue			:= FALSE;

		eChgPage			:= UIP0931ConvInv;

	ELSIF tyP0920MtrNPneuCtrl.tyMtrNPneuCtrl.tyBtnAW.bRtCompl = TRUE THEN
		tyP0920MtrNPneuCtrl.tyMtrNPneuCtrl.tyBtnAW.bRtCompl			:= FALSE;
		tyP0920MtrNPneuCtrl.tyMtrNPneuCtrl.tyBtnAW.bValue			:= FALSE;

		eChgPage			:= UIP0934AW;

	ELSIF tyP0920MtrNPneuCtrl.tyMtrNPneuCtrl.tyBtnClampNoRS.bRtCompl = TRUE THEN
		tyP0920MtrNPneuCtrl.tyMtrNPneuCtrl.tyBtnClampNoRS.bRtCompl		:= FALSE;
		tyP0920MtrNPneuCtrl.tyMtrNPneuCtrl.tyBtnClampNoRS.bValue		:= FALSE;

		eChgPage			:= UIP0921ClampNoRS;

	ELSIF tyP0920MtrNPneuCtrl.tyMtrNPneuCtrl.tyBtnClampWithRS.bRtCompl = TRUE THEN
		tyP0920MtrNPneuCtrl.tyMtrNPneuCtrl.tyBtnClampWithRS.bRtCompl	:= FALSE;
		tyP0920MtrNPneuCtrl.tyMtrNPneuCtrl.tyBtnClampWithRS.bValue		:= FALSE;

		eChgPage			:= UIP0924ClampWithRS;

	ELSIF tyP0920MtrNPneuCtrl.tyMtrNPneuCtrl.tyBtnShutter.bRtCompl = TRUE THEN
		tyP0920MtrNPneuCtrl.tyMtrNPneuCtrl.tyBtnShutter.bRtCompl	:= FALSE;
		tyP0920MtrNPneuCtrl.tyMtrNPneuCtrl.tyBtnShutter.bValue		:= FALSE;

		eChgPage			:= UIP0922Shutter;

	END_IF

END_ACTION
```

#### Act_EntP0921Disp.st
```iecst
ACTION Act_EntP0921Disp:

	p_tyC0002FullMask ACCESS ADR(tyP0921ClampNoRS.tyFullMaskHide);

	p_tyC0004Navi ACCESS ADR(tyP0921ClampNoRS.tyNaviBack);

	p_tyC0005Main ACCESS ADR(tyCommon.tyMain);

	p_tyC0007Notif ACCESS ADR(tyCommon.tyNotif);

	p_tyC0008MsgBox ACCESS ADR(tyP0921ClampNoRS.tyMsgBoxHide);

	p_tyC0009Info ACCESS ADR(tyCommon.tyInfo);

	p_tyC0011Loading ACCESS ADR(tyCommon.tyLoading);

	p_tyP0921ClampNoRSCom ACCESS ADR(tyP0921ClampNoRS.tyCom);

	p_tyP0921ClampNoRSDC ACCESS ADR(tyP0921ClampNoRS.tyDC);

	p_tyP0921ClampNoRSFB ACCESS ADR(tyP0921ClampNoRS.tyFB);

	//Display
	IF tyP0921ClampNoRS.tyCom.tyBtnDCCtrl.bValue = TRUE THEN
		fUIInRtStatOff(ADR(tyP0921ClampNoRS.tyDC.tyLyr.uiRtStat));
		fUIInRtStatHide(ADR(tyP0921ClampNoRS.tyFB.tyLyr.uiRtStat));
	ELSE
		fUIInRtStatHide(ADR(tyP0921ClampNoRS.tyDC.tyLyr.uiRtStat));
		fUIInRtStatOff(ADR(tyP0921ClampNoRS.tyFB.tyLyr.uiRtStat));
	END_IF

END_ACTION
```

#### Act_OptP0921FullMask.st
```iecst
ACTION Act_OptP0921FullMask:

	IF eCurrPage = UIP0921ClampNoRS THEN

		IF p_tyDI.bEStopSig = FALSE THEN
			p_tyC0002FullMask ACCESS ADR(tyP0921ClampNoRS.tyFullMaskEStop);

		ELSIF p_tyDI.bCoverSWSig = FALSE THEN
			p_tyC0002FullMask ACCESS ADR(tyP0921ClampNoRS.tyFullMaskCWSig);

		ELSIF p_tyDI.bSafetyRlySig = FALSE THEN
			p_tyC0002FullMask ACCESS ADR(tyP0921ClampNoRS.tyFullMaskSafetyRly);

		ELSE
			p_tyC0002FullMask ACCESS ADR(tyP0921ClampNoRS.tyFullMaskHide);

		END_IF

	END_IF

END_ACTION
```

#### Act_OptP0921Navi.st
```iecst
ACTION Act_OptP0921Navi:

	IF tyP0921ClampNoRS.tyNaviBack.tyBtnBack.bRtCompl = TRUE THEN
		tyP0921ClampNoRS.tyNaviBack.tyBtnBack.bRtCompl 	:= FALSE;
		tyP0921ClampNoRS.tyNaviBack.tyBtnBack.bValue		:= FALSE;

		eChgPage	:= UIP0920MtrNPneuCtrl;

	END_IF

END_ACTION
```

#### Act_OptP0921ChgLyr.st
```iecst
ACTION Act_OptP0921ChgLyr:

	IF tyP0921ClampNoRS.tyCom.tyBtnDCCtrl.bRtCompl = TRUE THEN
		tyP0921ClampNoRS.tyCom.tyBtnDCCtrl.bRtCompl := FALSE;

		IF tyP0921ClampNoRS.tyCom.tyBtnDCCtrl.bValue = TRUE THEN
			fUIInRtStatOff(ADR(tyP0921ClampNoRS.tyDC.tyLyr.uiRtStat));
			fUIInRtStatHide(ADR(tyP0921ClampNoRS.tyFB.tyLyr.uiRtStat));
		ELSE
			fUIInRtStatHide(ADR(tyP0921ClampNoRS.tyDC.tyLyr.uiRtStat));
			fUIInRtStatOff(ADR(tyP0921ClampNoRS.tyFB.tyLyr.uiRtStat));
		END_IF
	END_IF

END_ACTION
```

#### Act_OptP0921UpdtData.st
```iecst
ACTION Act_OptP0921UpdtData:

	//Update Bitmap
	IF p_bClampExtCtrl THEN
		tyP0921ClampNoRS.tyCom.tyBitmapMc.usiValueIdx	:= 1;
	ELSE
		tyP0921ClampNoRS.tyCom.tyBitmapMc.usiValueIdx	:= 0;
	END_IF

END_ACTION
```

#### Act_OptP0921FBCtrl.st
```iecst
ACTION Act_OptP0921FBCtrl:

	IF tyP0921ClampNoRS.tyCom.tyBtnDCCtrl.bValue = FALSE THEN

		IF tyP0921ClampNoRS.tyFB.tyBtnRet.bRtCompl = TRUE THEN
			tyP0921ClampNoRS.tyFB.tyBtnRet.bRtCompl	:= FALSE;

			tyP0921ClampNoRS.tyFB.tyBtnRet.bValue		:= TRUE;
			tyP0921ClampNoRS.tyFB.tyBtnExt.bValue		:= FALSE;

		ELSIF tyP0921ClampNoRS.tyFB.tyBtnExt.bRtCompl = TRUE THEN
			tyP0921ClampNoRS.tyFB.tyBtnExt.bRtCompl	:= FALSE;

			tyP0921ClampNoRS.tyFB.tyBtnExt.bValue		:= TRUE;
			tyP0921ClampNoRS.tyFB.tyBtnRet.bValue		:= FALSE;
		END_IF

		IF tyP0921ClampNoRS.tyFB.tyBtnRet.bValue = TRUE THEN
			eClampAct	:= PneuActRet;

			IF p_eClampStat = PneuActRet AND p_eClampStatus = Done THEN
				eClampAct	:= PneuActIdle;

				tyP0921ClampNoRS.tyCom.tyBitmapMc.usiValueIdx	:= 0;
				tyP0921ClampNoRS.tyFB.tyBtnRet.bValue	:= FALSE;

			ELSIF p_eClampStatus = Error THEN

				tyP0921ClampNoRS.tyFB.tyBtnRet.bValue	:= FALSE;
			END_IF

		ELSIF tyP0921ClampNoRS.tyFB.tyBtnExt.bValue = TRUE THEN
			eClampAct	:= PneuActExt;

			IF p_eClampStat = PneuActExt AND p_eClampStatus = Done THEN
				eClampAct	:= PneuActIdle;

				tyP0921ClampNoRS.tyCom.tyBitmapMc.usiValueIdx	:= 1;
				tyP0921ClampNoRS.tyFB.tyBtnExt.bValue := FALSE;

			ELSIF p_eClampStatus = Error THEN

				tyP0921ClampNoRS.tyFB.tyBtnExt.bValue := FALSE;
			END_IF
		END_IF

		//Update Direct Control Status

		tyP0921ClampNoRS.tyDC.tyBtnRet.bRtCompl		:= FALSE;
		tyP0921ClampNoRS.tyDC.tyBtnExt.bRtCompl		:= FALSE;
		tyP0921ClampNoRS.tyDC.tyBtnRet.bValue		:= p_bClampRetCtrl;
		tyP0921ClampNoRS.tyDC.tyBtnExt.bValue		:= p_bClampExtCtrl;

		IF p_tyUsrMgmtCurrAccessRgt.bManualFBOnly THEN
			fUIInRtStatOff(ADR(tyP0921ClampNoRS.tyCom.tyBtnDCCtrl.uiMaskRtStat));
		ELSE
			fUIInRtStatHide(ADR(tyP0921ClampNoRS.tyCom.tyBtnDCCtrl.uiMaskRtStat));

		END_IF

	END_IF

END_ACTION
```

#### Act_OptP0921FBStat.st
```iecst
ACTION Act_OptP0921FBStat:

	tyP0921ClampNoRS.tyFB.tyStringStat.sValue	:= p_sClampStatTxt;

END_ACTION
```

#### Act_OptP0921DCCtrl.st
```iecst
ACTION Act_OptP0921DCCtrl:

	IF tyP0921ClampNoRS.tyCom.tyBtnDCCtrl.bValue = TRUE THEN

		IF p_bClampTwoCtrlOut = FALSE THEN

			IF tyP0921ClampNoRS.tyDC.tyBtnRet.bRtCompl = TRUE THEN
				tyP0921ClampNoRS.tyDC.tyBtnRet.bValue	:= TRUE;
				tyP0921ClampNoRS.tyDC.tyBtnExt.bValue	:= FALSE;

				eClampAct	:= PneuActSetRet;

				IF p_eClampStat = PneuActSetRet AND p_eClampStatus = Done THEN
					eClampAct	:= PneuActIdle;

					tyP0921ClampNoRS.tyCom.tyBitmapMc.usiValueIdx	:= 0;
					tyP0921ClampNoRS.tyDC.tyBtnRet.bRtCompl	:= FALSE;
				END_IF

			ELSIF tyP0921ClampNoRS.tyDC.tyBtnExt.bRtCompl = TRUE THEN
				tyP0921ClampNoRS.tyDC.tyBtnExt.bValue	:= TRUE;
				tyP0921ClampNoRS.tyDC.tyBtnRet.bValue	:= FALSE;

				eClampAct	:= PneuActSetExt;

				IF p_eClampStat = PneuActSetExt AND p_eClampStatus = Done THEN
					eClampAct	:= PneuActIdle;

					tyP0921ClampNoRS.tyCom.tyBitmapMc.usiValueIdx	:= 1;
					tyP0921ClampNoRS.tyDC.tyBtnExt.bRtCompl	:= FALSE;
				END_IF

			END_IF

		ELSE

			IF (tyP0921ClampNoRS.tyDC.tyBtnRet.bRtCompl = TRUE) OR (tyP0921ClampNoRS.tyDC.tyBtnExt.bRtCompl = TRUE) THEN

				IF (tyP0921ClampNoRS.tyDC.tyBtnRet.bValue = TRUE) AND (tyP0921ClampNoRS.tyDC.tyBtnExt.bValue = TRUE) THEN
					eClampAct	:= PneuActSetAll;

					IF p_eClampStat = PneuActSetAll AND p_eClampStatus = Done THEN
						eClampAct	:= PneuActIdle;

						tyP0921ClampNoRS.tyDC.tyBtnRet.bRtCompl	:= FALSE;
						tyP0921ClampNoRS.tyDC.tyBtnExt.bRtCompl	:= FALSE;
					END_IF

				ELSIF (tyP0921ClampNoRS.tyDC.tyBtnRet.bValue = TRUE) AND (tyP0921ClampNoRS.tyDC.tyBtnExt.bValue = FALSE) THEN
					eClampAct	:= PneuActSetRet;

					IF p_eClampStat = PneuActSetRet AND p_eClampStatus = Done THEN
						eClampAct	:= PneuActIdle;

						tyP0921ClampNoRS.tyCom.tyBitmapMc.usiValueIdx	:= 0;
						tyP0921ClampNoRS.tyDC.tyBtnRet.bRtCompl	:= FALSE;
						tyP0921ClampNoRS.tyDC.tyBtnExt.bRtCompl	:= FALSE;
					END_IF

				ELSIF (tyP0921ClampNoRS.tyDC.tyBtnRet.bValue = FALSE) AND (tyP0921ClampNoRS.tyDC.tyBtnExt.bValue = TRUE) THEN
					eClampAct	:= PneuActSetExt;

					IF p_eClampStat = PneuActSetExt AND p_eClampStatus = Done THEN
						eClampAct	:= PneuActIdle;

						tyP0921ClampNoRS.tyCom.tyBitmapMc.usiValueIdx	:= 1;
						tyP0921ClampNoRS.tyDC.tyBtnRet.bRtCompl	:= FALSE;
						tyP0921ClampNoRS.tyDC.tyBtnExt.bRtCompl	:= FALSE;
					END_IF

				ELSE
					eClampAct	:= PneuActRstAll;

					IF p_eClampStat = PneuActRstAll AND p_eClampStatus = Done THEN
						eClampAct	:= PneuActIdle;

						tyP0921ClampNoRS.tyDC.tyBtnRet.bRtCompl	:= FALSE;
						tyP0921ClampNoRS.tyDC.tyBtnExt.bRtCompl	:= FALSE;
					END_IF

				END_IF

			END_IF

		END_IF

		tyP0921ClampNoRS.tyFB.tyBtnExt.bRtCompl	:= FALSE;
		tyP0921ClampNoRS.tyFB.tyBtnExt.bValue		:= FALSE;
		tyP0921ClampNoRS.tyFB.tyBtnRet.bRtCompl	:= FALSE;
		tyP0921ClampNoRS.tyFB.tyBtnRet.bValue		:= FALSE;

	END_IF

END_ACTION
```

#### Act_OptP0921RstMnl.st
```iecst
ACTION Act_OptP0921RstMnl:

	IF EDGEPOS(p_eClampStatus = Error) THEN

		eClampAct	:= PneuActIdle;

		tyP0921ClampNoRS.tyDC.tyBtnRet.bRtCompl		:= FALSE;
		tyP0921ClampNoRS.tyDC.tyBtnRet.bValue		:= FALSE;
		tyP0921ClampNoRS.tyDC.tyBtnExt.bRtCompl		:= FALSE;
		tyP0921ClampNoRS.tyDC.tyBtnExt.bValue		:= FALSE;

		tyP0921ClampNoRS.tyFB.tyBtnRet.bRtCompl		:= FALSE;
		tyP0921ClampNoRS.tyFB.tyBtnRet.bValue		:= FALSE;
		tyP0921ClampNoRS.tyFB.tyBtnExt.bRtCompl		:= FALSE;
		tyP0921ClampNoRS.tyFB.tyBtnExt.bValue		:= FALSE;

	END_IF

	IF EDGEPOS(bManualMod = FALSE) THEN

		tyP0921ClampNoRS.tyCom.tyBtnDCCtrl.bValue		:= FALSE;

		fUIInRtStatHide(ADR(tyP0921ClampNoRS.tyDC.tyLyr.uiRtStat));
		fUIInRtStatOff(ADR(tyP0921ClampNoRS.tyFB.tyLyr.uiRtStat));

		eClampAct	:= PneuActIdle;

		tyP0921ClampNoRS.tyDC.tyBtnRet.bRtCompl		:= FALSE;
		tyP0921ClampNoRS.tyDC.tyBtnRet.bValue		:= FALSE;
		tyP0921ClampNoRS.tyDC.tyBtnExt.bRtCompl		:= FALSE;
		tyP0921ClampNoRS.tyDC.tyBtnExt.bValue		:= FALSE;

		tyP0921ClampNoRS.tyFB.tyBtnRet.bRtCompl		:= FALSE;
		tyP0921ClampNoRS.tyFB.tyBtnRet.bValue		:= FALSE;
		tyP0921ClampNoRS.tyFB.tyBtnExt.bRtCompl		:= FALSE;
		tyP0921ClampNoRS.tyFB.tyBtnExt.bValue		:= FALSE;

	END_IF

END_ACTION
```

#### Act_EntP0922Disp.st
```iecst
ACTION Act_EntP0922Disp:

	//Access Address
	p_tyC0003DualMask ACCESS ADR(tyP0922InletNOutletShutter.tyDualMaskHide);

	p_tyC0004Navi ACCESS ADR(tyP0922InletNOutletShutter.tyNaviBack);

	p_tyC0005Main ACCESS ADR(tyCommon.tyMain);

	p_tyC0007Notif ACCESS ADR(tyCommon.tyNotif);

	p_tyC0008MsgBox ACCESS ADR(tyP0922InletNOutletShutter.tyMsgBoxHide);

	p_tyC0009Info ACCESS ADR(tyCommon.tyInfo);

	p_tyP0922InletShutterCom ACCESS ADR(tyP0922InletNOutletShutter.tyInletShutterCom);
	p_tyP0922InletShutterDC ACCESS ADR(tyP0922InletNOutletShutter.tyInletShutterDC);
	p_tyP0922InletShutterFB ACCESS ADR(tyP0922InletNOutletShutter.tyInletShutterFB);
	p_tyP0922InletShutterDis ACCESS ADR(tyP0922InletNOutletShutter.tyInletShutterDis);

	p_tyP0922OutletShutterCom ACCESS ADR(tyP0922InletNOutletShutter.tyOutletShutterCom);
	p_tyP0922OutletShutterDC ACCESS ADR(tyP0922InletNOutletShutter.tyOutletShutterDC);
	p_tyP0922OutletShutterFB ACCESS ADR(tyP0922InletNOutletShutter.tyOutletShutterFB);
	p_tyP0922OutletShutterDis ACCESS ADR(tyP0922InletNOutletShutter.tyOutletShutterDis);

	//Display
	tyP0922InletNOutletShutter.tyInletShutterDis.tyLyr.uiRtStat.0	:= NOT(p_tyNtParamCurr.bProjInletShutPrep AND p_tyMcParamCurr.bInShutterDis);

	//Display
	IF tyP0922InletNOutletShutter.tyInletShutterCom.tyBtnSwitch.bValue = TRUE THEN
		fUIInRtStatOff(ADR(tyP0922InletNOutletShutter.tyInletShutterDC.tyLyr.uiRtStat));
		fUIInRtStatHide(ADR(tyP0922InletNOutletShutter.tyInletShutterFB.tyLyr.uiRtStat));
	ELSE
		fUIInRtStatOff(ADR(tyP0922InletNOutletShutter.tyInletShutterFB.tyLyr.uiRtStat));
		fUIInRtStatHide(ADR(tyP0922InletNOutletShutter.tyInletShutterDC.tyLyr.uiRtStat));
	END_IF

	IF tyP0922InletNOutletShutter.tyOutletShutterCom.tyBtnSwitch.bValue = TRUE THEN
		fUIInRtStatOff(ADR(tyP0922InletNOutletShutter.tyOutletShutterDC.tyLyr.uiRtStat));
		fUIInRtStatHide(ADR(tyP0922InletNOutletShutter.tyOutletShutterFB.tyLyr.uiRtStat));
	ELSE
		fUIInRtStatOff(ADR(tyP0922InletNOutletShutter.tyOutletShutterFB.tyLyr.uiRtStat));
		fUIInRtStatHide(ADR(tyP0922InletNOutletShutter.tyOutletShutterDC.tyLyr.uiRtStat));
	END_IF

END_ACTION
```

#### Act_OptP0922Navi.st
```iecst
ACTION Act_OptP0922Navi:

	IF tyP0922InletNOutletShutter.tyNaviBack.tyBtnBack.bRtCompl = TRUE THEN
		eChgPage		:= UIP0920MtrNPneuCtrl;

		tyP0922InletNOutletShutter.tyNaviBack.tyBtnBack.bRtCompl 	:= FALSE;
		tyP0922InletNOutletShutter.tyNaviBack.tyBtnBack.bValue		:= FALSE;
	END_IF

END_ACTION
```

#### Act_OptP0922DualMask.st
```iecst
ACTION Act_OptP0922DualMask:

	IF eCurrPage = UIP0922Shutter THEN

		IF p_tyDI.bEStopSig = FALSE THEN
			p_tyC0003DualMask ACCESS ADR(tyP0922InletNOutletShutter.tyDualMaskEStop);

			tyP0922InletNOutletShutter.tyDualMaskEStop.tyBtnLeftMask.uiMaskRtStat.0	:= NOT p_tyNtParamCurr.bProjInletShutPrep;
			tyP0922InletNOutletShutter.tyDualMaskEStop.tyBtnRgtMask.uiMaskRtStat.0	:= NOT p_tyNtParamCurr.bProjOutletShutPrep;

		ELSIF p_tyDI.bCoverSWSig = FALSE THEN
			p_tyC0003DualMask ACCESS ADR(tyP0922InletNOutletShutter.tyDualMaskCWSig);

			tyP0922InletNOutletShutter.tyDualMaskCWSig.tyBtnLeftMask.uiMaskRtStat.0	:= NOT p_tyNtParamCurr.bProjInletShutPrep;
			tyP0922InletNOutletShutter.tyDualMaskCWSig.tyBtnRgtMask.uiMaskRtStat.0	:= NOT p_tyNtParamCurr.bProjOutletShutPrep;

		ELSIF p_tyDI.bSafetyRlySig = FALSE THEN
			p_tyC0003DualMask ACCESS ADR(tyP0922InletNOutletShutter.tyDualMaskSafetyRly);

			tyP0922InletNOutletShutter.tyDualMaskSafetyRly.tyBtnLeftMask.uiMaskRtStat.0	:= NOT p_tyNtParamCurr.bProjInletShutPrep;
			tyP0922InletNOutletShutter.tyDualMaskSafetyRly.tyBtnRgtMask.uiMaskRtStat.0	:= NOT p_tyNtParamCurr.bProjOutletShutPrep;

		ELSIF p_eAWOpenStatus = Busy THEN
			p_tyC0003DualMask ACCESS ADR(tyP0922InletNOutletShutter.tyDualMaskAWMovInterrupt);

			tyP0922InletNOutletShutter.tyDualMaskAWMovInterrupt.tyBtnLeftMask.uiMaskRtStat.0	:= NOT p_tyNtParamCurr.bProjInletShutPrep;
			tyP0922InletNOutletShutter.tyDualMaskAWMovInterrupt.tyBtnRgtMask.uiMaskRtStat.0		:= NOT p_tyNtParamCurr.bProjOutletShutPrep;

		ELSE
			p_tyC0003DualMask ACCESS ADR(tyP0922InletNOutletShutter.tyDualMaskHide);

		END_IF

	END_IF

END_ACTION
```

#### Act_OptP0922InletShutterChgLyr.st
```iecst
ACTION Act_OptP0922InletShutterChgLyr:

	IF tyP0922InletNOutletShutter.tyInletShutterCom.tyBtnSwitch.bRtCompl THEN
		tyP0922InletNOutletShutter.tyInletShutterCom.tyBtnSwitch.bRtCompl := FALSE;

		IF tyP0922InletNOutletShutter.tyInletShutterCom.tyBtnSwitch.bValue = TRUE THEN
			fUIInRtStatOff(ADR(tyP0922InletNOutletShutter.tyInletShutterDC.tyLyr.uiRtStat));
			fUIInRtStatHide(ADR(tyP0922InletNOutletShutter.tyInletShutterFB.tyLyr.uiRtStat));
		ELSE
			fUIInRtStatHide(ADR(tyP0922InletNOutletShutter.tyInletShutterDC.tyLyr.uiRtStat));
			fUIInRtStatOff(ADR(tyP0922InletNOutletShutter.tyInletShutterFB.tyLyr.uiRtStat));
		END_IF

	END_IF

END_ACTION
```

#### Act_OptP0922InletShutterSen.st
```iecst
ACTION Act_OptP0922InletShutterSen:

	tyP0922InletNOutletShutter.tyInletShutterCom.tyBtnOpenRS.bValue		:= p_tyDI.bInShutterOpenRS;
	tyP0922InletNOutletShutter.tyInletShutterCom.tyBtnCloseRS.bValue	:= p_tyDI.bInShutterCloseRS;

	//Machine Bitmap
	IF p_tyDI.bInShutterOpenRS = TRUE THEN
		IF p_tyNtParamCurr.tyDOSettings.diTLGreen<>0 OR p_tyNtParamCurr.tyDOSettings.diTLAmber<>0 OR p_tyNtParamCurr.tyDOSettings.diTLRed<>0 THEN
			IF p_tyNtParamCurr.eTLBuzMode=TLBuzModBHTC THEN
				tyP0922InletNOutletShutter.tyInletShutterCom.tyBitmapMc.usiValueIdx	:= 200;
			ELSE
				tyP0922InletNOutletShutter.tyInletShutterCom.tyBitmapMc.usiValueIdx	:= 100;
			END_IF
		ELSE
			tyP0922InletNOutletShutter.tyInletShutterCom.tyBitmapMc.usiValueIdx	:= 0;
		END_IF
	ELSE
		IF p_tyNtParamCurr.tyDOSettings.diTLGreen<>0 OR p_tyNtParamCurr.tyDOSettings.diTLAmber<>0 OR p_tyNtParamCurr.tyDOSettings.diTLRed<>0 THEN
			IF p_tyNtParamCurr.eTLBuzMode=TLBuzModBHTC THEN
				tyP0922InletNOutletShutter.tyInletShutterCom.tyBitmapMc.usiValueIdx	:= 201;
			ELSE
				tyP0922InletNOutletShutter.tyInletShutterCom.tyBitmapMc.usiValueIdx	:= 101;
			END_IF
		ELSE
			tyP0922InletNOutletShutter.tyInletShutterCom.tyBitmapMc.usiValueIdx	:= 1;
		END_IF
	END_IF

END_ACTION
```

#### Act_OptP0922InletShutterFB.st
```iecst
ACTION Act_OptP0922InletShutterFB:

	IF tyP0922InletNOutletShutter.tyInletShutterCom.tyBtnSwitch.bValue = FALSE THEN

		IF tyP0922InletNOutletShutter.tyInletShutterFB.tyBtnOpen.bRtCompl = TRUE THEN
			tyP0922InletNOutletShutter.tyInletShutterFB.tyBtnOpen.bRtCompl	:= FALSE;

			tyP0922InletNOutletShutter.tyInletShutterFB.tyBtnOpen.bValue	:= TRUE;
			tyP0922InletNOutletShutter.tyInletShutterFB.tyBtnClose.bValue	:= FALSE;

		ELSIF tyP0922InletNOutletShutter.tyInletShutterFB.tyBtnClose.bRtCompl = TRUE THEN
			tyP0922InletNOutletShutter.tyInletShutterFB.tyBtnClose.bRtCompl	:= FALSE;

			tyP0922InletNOutletShutter.tyInletShutterFB.tyBtnClose.bValue	:= TRUE;
			tyP0922InletNOutletShutter.tyInletShutterFB.tyBtnOpen.bValue	:= FALSE;
		END_IF

		IF tyP0922InletNOutletShutter.tyInletShutterFB.tyBtnOpen.bValue = TRUE THEN
			eInShutterAct	:= PneuActRet;

			IF p_eInShutterStat = PneuActRet AND p_eInShutterStatus = Done THEN
				eInShutterAct	:= PneuActIdle;

				tyP0922InletNOutletShutter.tyInletShutterFB.tyBtnOpen.bValue	:= FALSE;
			ELSIF p_eInShutterStatus = Error THEN
				tyP0922InletNOutletShutter.tyInletShutterFB.tyBtnOpen.bValue	:= FALSE;
			END_IF

		ELSIF tyP0922InletNOutletShutter.tyInletShutterFB.tyBtnClose.bValue = TRUE THEN
			eInShutterAct	:= PneuActExt;

			IF p_eInShutterStat = PneuActExt AND p_eInShutterStatus = Done THEN
				eInShutterAct	:= PneuActIdle;

				tyP0922InletNOutletShutter.tyInletShutterFB.tyBtnClose.bValue := FALSE;
			ELSIF p_eInShutterStatus = Error THEN
				tyP0922InletNOutletShutter.tyInletShutterFB.tyBtnClose.bValue := FALSE;
			END_IF
		END_IF

		//Update Direct Control Status
		tyP0922InletNOutletShutter.tyInletShutterDC.tyBtnOpen.bRtCompl	:= FALSE;
		tyP0922InletNOutletShutter.tyInletShutterDC.tyBtnClose.bRtCompl	:= FALSE;
		tyP0922InletNOutletShutter.tyInletShutterDC.tyBtnOpen.bValue	:= p_bInShutterRetCtrl;
		tyP0922InletNOutletShutter.tyInletShutterDC.tyBtnClose.bValue	:= p_bInShutterExtCtrl;

		IF p_tyUsrMgmtCurrAccessRgt.bManualFBOnly THEN
			fUIInRtStatOff(ADR(tyP0922InletNOutletShutter.tyInletShutterCom.tyBtnSwitch.uiMaskRtStat));
		ELSE
			fUIInRtStatHide(ADR(tyP0922InletNOutletShutter.tyInletShutterCom.tyBtnSwitch.uiMaskRtStat));

		END_IF

	END_IF

END_ACTION
```

#### Act_OptP0922InletShutterFBStat.st
```iecst
ACTION Act_OptP0922InletShutterFBStat:

	tyP0922InletNOutletShutter.tyInletShutterFB.tyStringStat.sValue	:= p_sInShutterStatTxt;

END_ACTION
```

#### Act_OptP0922InletShutterDC.st
```iecst
ACTION Act_OptP0922InletShutterDC:

	IF tyP0922InletNOutletShutter.tyInletShutterCom.tyBtnSwitch.bValue = TRUE THEN
		IF p_bInShutterTwoCtrlOut = FALSE THEN
			IF tyP0922InletNOutletShutter.tyInletShutterDC.tyBtnOpen.bRtCompl = TRUE THEN
				tyP0922InletNOutletShutter.tyInletShutterDC.tyBtnOpen.bValue	:= TRUE;
				tyP0922InletNOutletShutter.tyInletShutterDC.tyBtnClose.bValue	:= FALSE;

				eInShutterAct	:= PneuActSetRet;

				IF p_eInShutterStat = PneuActSetRet AND p_eInShutterStatus = Done THEN
					eInShutterAct	:= PneuActIdle;

					tyP0922InletNOutletShutter.tyInletShutterDC.tyBtnOpen.bRtCompl	:= FALSE;
				END_IF

			ELSIF tyP0922InletNOutletShutter.tyInletShutterDC.tyBtnClose.bRtCompl = TRUE THEN
				tyP0922InletNOutletShutter.tyInletShutterDC.tyBtnClose.bValue	:= TRUE;
				tyP0922InletNOutletShutter.tyInletShutterDC.tyBtnOpen.bValue	:= FALSE;

				eInShutterAct	:= PneuActSetExt;

				IF p_eInShutterStat = PneuActSetExt AND p_eInShutterStatus = Done THEN
					eInShutterAct	:= PneuActIdle;

					tyP0922InletNOutletShutter.tyInletShutterDC.tyBtnClose.bRtCompl	:= FALSE;
				END_IF
			END_IF

		ELSE
			IF (tyP0922InletNOutletShutter.tyInletShutterDC.tyBtnOpen.bRtCompl = TRUE) OR (tyP0922InletNOutletShutter.tyInletShutterDC.tyBtnClose.bRtCompl = TRUE) THEN
				IF (tyP0922InletNOutletShutter.tyInletShutterDC.tyBtnOpen.bValue = TRUE) AND (tyP0922InletNOutletShutter.tyInletShutterDC.tyBtnClose.bValue = TRUE) THEN
					eInShutterAct	:= PneuActSetAll;

					IF p_eInShutterStat = PneuActSetAll AND p_eInShutterStatus = Done THEN
						eInShutterAct	:= PneuActIdle;

						tyP0922InletNOutletShutter.tyInletShutterDC.tyBtnOpen.bRtCompl	:= FALSE;
						tyP0922InletNOutletShutter.tyInletShutterDC.tyBtnClose.bRtCompl	:= FALSE;
					END_IF

				ELSIF (tyP0922InletNOutletShutter.tyInletShutterDC.tyBtnOpen.bValue = TRUE) AND (tyP0922InletNOutletShutter.tyInletShutterDC.tyBtnClose.bValue = FALSE) THEN
					eInShutterAct	:= PneuActSetRet;

					IF p_eInShutterStat = PneuActSetRet AND p_eInShutterStatus = Done THEN
						eInShutterAct	:= PneuActIdle;

						tyP0922InletNOutletShutter.tyInletShutterDC.tyBtnOpen.bRtCompl	:= FALSE;
						tyP0922InletNOutletShutter.tyInletShutterDC.tyBtnClose.bRtCompl	:= FALSE;
					END_IF

				ELSIF (tyP0922InletNOutletShutter.tyInletShutterDC.tyBtnOpen.bValue = FALSE) AND (tyP0922InletNOutletShutter.tyInletShutterDC.tyBtnClose.bValue = TRUE) THEN
					eInShutterAct	:= PneuActSetExt;

					IF p_eInShutterStat = PneuActSetExt AND p_eInShutterStatus = Done THEN
						eInShutterAct	:= PneuActIdle;

						tyP0922InletNOutletShutter.tyInletShutterDC.tyBtnOpen.bRtCompl	:= FALSE;
						tyP0922InletNOutletShutter.tyInletShutterDC.tyBtnClose.bRtCompl	:= FALSE;
					END_IF

				ELSE
					eInShutterAct	:= PneuActRstAll;

					IF p_eInShutterStat = PneuActRstAll AND p_eInShutterStatus = Done THEN
						eInShutterAct	:= PneuActIdle;

						tyP0922InletNOutletShutter.tyInletShutterDC.tyBtnOpen.bRtCompl	:= FALSE;
						tyP0922InletNOutletShutter.tyInletShutterDC.tyBtnClose.bRtCompl	:= FALSE;
					END_IF

				END_IF
			END_IF
		END_IF

		tyP0922InletNOutletShutter.tyInletShutterFB.tyBtnClose.bRtCompl	:= FALSE;
		tyP0922InletNOutletShutter.tyInletShutterFB.tyBtnClose.bValue	:= FALSE;
		tyP0922InletNOutletShutter.tyInletShutterFB.tyBtnOpen.bRtCompl	:= FALSE;
		tyP0922InletNOutletShutter.tyInletShutterFB.tyBtnOpen.bValue	:= FALSE;

	END_IF

END_ACTION
```

#### Act_OptP0922OutletShutterChgLyr.st
```iecst
ACTION Act_OptP0922OutletShutterChgLyr:

	IF	tyP0922InletNOutletShutter.tyOutletShutterCom.tyBtnSwitch.bRtCompl THEN
			tyP0922InletNOutletShutter.tyOutletShutterCom.tyBtnSwitch.bRtCompl := FALSE;

		IF tyP0922InletNOutletShutter.tyOutletShutterCom.tyBtnSwitch.bValue = TRUE THEN
			fUIInRtStatOff(ADR(tyP0922InletNOutletShutter.tyOutletShutterDC.tyLyr.uiRtStat));
			fUIInRtStatHide(ADR(tyP0922InletNOutletShutter.tyOutletShutterFB.tyLyr.uiRtStat));
		ELSE
			fUIInRtStatHide(ADR(tyP0922InletNOutletShutter.tyOutletShutterDC.tyLyr.uiRtStat));
			fUIInRtStatOff(ADR(tyP0922InletNOutletShutter.tyOutletShutterFB.tyLyr.uiRtStat));
		END_IF

	END_IF

END_ACTION
```

#### Act_OptP0922OutletShutterSen.st
```iecst
ACTION Act_OptP0922OutletShutterSen:

	tyP0922InletNOutletShutter.tyOutletShutterCom.tyBtnOpenRS.bValue	:= p_tyDI.bOutShutterOpenRS;
	tyP0922InletNOutletShutter.tyOutletShutterCom.tyBtnCloseRS.bValue	:= p_tyDI.bOutShutterCloseRS;

	//Machine Bitmap
	IF p_tyDI.bOutShutterOpenRS = TRUE THEN
		IF p_tyNtParamCurr.tyDOSettings.diTLGreen<>0 OR p_tyNtParamCurr.tyDOSettings.diTLAmber<>0 OR p_tyNtParamCurr.tyDOSettings.diTLRed<>0 THEN
			IF p_tyNtParamCurr.eTLBuzMode=TLBuzModBHTC THEN
				tyP0922InletNOutletShutter.tyOutletShutterCom.tyBitmapMc.usiValueIdx	:= 200;
			ELSE
				tyP0922InletNOutletShutter.tyOutletShutterCom.tyBitmapMc.usiValueIdx	:= 100;
			END_IF
		ELSE
			tyP0922InletNOutletShutter.tyOutletShutterCom.tyBitmapMc.usiValueIdx	:= 0;
		END_IF
	ELSE
		IF p_tyNtParamCurr.tyDOSettings.diTLGreen<>0 OR p_tyNtParamCurr.tyDOSettings.diTLAmber<>0 OR p_tyNtParamCurr.tyDOSettings.diTLRed<>0 THEN
			IF p_tyNtParamCurr.eTLBuzMode=TLBuzModBHTC THEN
				tyP0922InletNOutletShutter.tyOutletShutterCom.tyBitmapMc.usiValueIdx	:= 201;
			ELSE
				tyP0922InletNOutletShutter.tyOutletShutterCom.tyBitmapMc.usiValueIdx	:= 101;
			END_IF
		ELSE
			tyP0922InletNOutletShutter.tyOutletShutterCom.tyBitmapMc.usiValueIdx	:= 1;
		END_IF
	END_IF

END_ACTION
```

#### Act_OptP0922OutletShutterFB.st
```iecst
ACTION Act_OptP0922OutletShutterFB:

	IF tyP0922InletNOutletShutter.tyOutletShutterCom.tyBtnSwitch.bValue = FALSE THEN
		// FB Control
		IF tyP0922InletNOutletShutter.tyOutletShutterFB.tyBtnOpen.bRtCompl = TRUE THEN
			tyP0922InletNOutletShutter.tyOutletShutterFB.tyBtnOpen.bRtCompl	:= FALSE;

			tyP0922InletNOutletShutter.tyOutletShutterFB.tyBtnOpen.bValue	:= TRUE;
			tyP0922InletNOutletShutter.tyOutletShutterFB.tyBtnClose.bValue	:= FALSE;

		ELSIF tyP0922InletNOutletShutter.tyOutletShutterFB.tyBtnClose.bRtCompl = TRUE THEN
			tyP0922InletNOutletShutter.tyOutletShutterFB.tyBtnClose.bRtCompl	:= FALSE;

			tyP0922InletNOutletShutter.tyOutletShutterFB.tyBtnClose.bValue	:= TRUE;
			tyP0922InletNOutletShutter.tyOutletShutterFB.tyBtnOpen.bValue	:= FALSE;
		END_IF

		IF tyP0922InletNOutletShutter.tyOutletShutterFB.tyBtnOpen.bValue = TRUE THEN
			eOutShutterAct	:= PneuActRet;

			IF p_eOutShutterStat = PneuActRet AND p_eOutShutterStatus = Done THEN
				eOutShutterAct	:= PneuActIdle;

				tyP0922InletNOutletShutter.tyOutletShutterFB.tyBtnOpen.bValue	:= FALSE;
			ELSIF p_eOutShutterStatus = Error THEN
				tyP0922InletNOutletShutter.tyOutletShutterFB.tyBtnOpen.bValue	:= FALSE;
			END_IF

		ELSIF tyP0922InletNOutletShutter.tyOutletShutterFB.tyBtnClose.bValue = TRUE THEN
			eOutShutterAct	:= PneuActExt;

			IF p_eOutShutterStat = PneuActExt AND p_eOutShutterStatus = Done THEN
				eOutShutterAct	:= PneuActIdle;

				tyP0922InletNOutletShutter.tyOutletShutterFB.tyBtnClose.bValue := FALSE;
			ELSIF p_eOutShutterStatus = Error THEN
				tyP0922InletNOutletShutter.tyOutletShutterFB.tyBtnClose.bValue := FALSE;
			END_IF
		END_IF

		//UpdateStatus
		tyP0922InletNOutletShutter.tyOutletShutterDC.tyBtnClose.bRtCompl	:= FALSE;
		tyP0922InletNOutletShutter.tyOutletShutterDC.tyBtnOpen.bRtCompl		:= FALSE;
		tyP0922InletNOutletShutter.tyOutletShutterDC.tyBtnClose.bValue		:= p_bOutShutterExtCtrl;
		tyP0922InletNOutletShutter.tyOutletShutterDC.tyBtnOpen.bValue		:= p_bOutShutterRetCtrl;

		IF p_tyUsrMgmtCurrAccessRgt.bManualFBOnly THEN
			fUIInRtStatOff(ADR(tyP0922InletNOutletShutter.tyOutletShutterCom.tyBtnSwitch.uiMaskRtStat));
		ELSE
			fUIInRtStatHide(ADR(tyP0922InletNOutletShutter.tyOutletShutterCom.tyBtnSwitch.uiMaskRtStat));
		END_IF
	END_IF

END_ACTION
```

#### Act_OptP0922OutletShutterFBStat.st
```iecst
ACTION Act_OptP0922OutletShutterFBStat:

	tyP0922InletNOutletShutter.tyOutletShutterFB.tyStringStat.sValue	:= p_sOutShutterStatTxt;

END_ACTION
```

#### Act_OptP0922OutletShutterDC.st
```iecst
ACTION Act_OptP0922OutletShutterDC:

	// Direct Control
	IF tyP0922InletNOutletShutter.tyOutletShutterCom.tyBtnSwitch.bValue = TRUE THEN
		IF p_bOutShutterTwoCtrlOut = FALSE THEN
			IF tyP0922InletNOutletShutter.tyOutletShutterDC.tyBtnOpen.bRtCompl = TRUE THEN
				tyP0922InletNOutletShutter.tyOutletShutterDC.tyBtnOpen.bValue	:= TRUE;
				tyP0922InletNOutletShutter.tyOutletShutterDC.tyBtnClose.bValue	:= FALSE;

				eOutShutterAct	:= PneuActSetRet;

				IF p_eOutShutterStat = PneuActSetRet AND p_eOutShutterStatus = Done THEN
					eOutShutterAct	:= PneuActIdle;

					tyP0922InletNOutletShutter.tyOutletShutterDC.tyBtnOpen.bRtCompl	:= FALSE;
				END_IF

			ELSIF tyP0922InletNOutletShutter.tyOutletShutterDC.tyBtnClose.bRtCompl = TRUE THEN
				tyP0922InletNOutletShutter.tyOutletShutterDC.tyBtnClose.bValue	:= TRUE;
				tyP0922InletNOutletShutter.tyOutletShutterDC.tyBtnOpen.bValue	:= FALSE;

				eOutShutterAct	:= PneuActSetExt;

				IF p_eOutShutterStat = PneuActSetExt AND p_eOutShutterStatus = Done THEN
					eOutShutterAct	:= PneuActIdle;

					tyP0922InletNOutletShutter.tyOutletShutterDC.tyBtnClose.bRtCompl	:= FALSE;
				END_IF
			END_IF

		ELSE
			IF (tyP0922InletNOutletShutter.tyOutletShutterDC.tyBtnOpen.bRtCompl = TRUE) OR (tyP0922InletNOutletShutter.tyOutletShutterDC.tyBtnClose.bRtCompl = TRUE) THEN
				IF (tyP0922InletNOutletShutter.tyOutletShutterDC.tyBtnOpen.bValue = TRUE) AND (tyP0922InletNOutletShutter.tyOutletShutterDC.tyBtnClose.bValue = TRUE) THEN
					eOutShutterAct	:= PneuActSetAll;

					IF p_eOutShutterStat = PneuActSetAll AND p_eOutShutterStatus = Done THEN
						eOutShutterAct	:= PneuActIdle;

						tyP0922InletNOutletShutter.tyOutletShutterDC.tyBtnOpen.bRtCompl		:= FALSE;
						tyP0922InletNOutletShutter.tyOutletShutterDC.tyBtnClose.bRtCompl	:= FALSE;
					END_IF

				ELSIF (tyP0922InletNOutletShutter.tyOutletShutterDC.tyBtnOpen.bValue = TRUE) AND (tyP0922InletNOutletShutter.tyOutletShutterDC.tyBtnClose.bValue = FALSE) THEN
					eOutShutterAct	:= PneuActSetRet;

					IF p_eOutShutterStat = PneuActSetRet AND p_eOutShutterStatus = Done THEN
						eOutShutterAct	:= PneuActIdle;

						tyP0922InletNOutletShutter.tyOutletShutterDC.tyBtnOpen.bRtCompl		:= FALSE;
						tyP0922InletNOutletShutter.tyOutletShutterDC.tyBtnClose.bRtCompl	:= FALSE;
					END_IF

				ELSIF (tyP0922InletNOutletShutter.tyOutletShutterDC.tyBtnOpen.bValue = FALSE) AND (tyP0922InletNOutletShutter.tyOutletShutterDC.tyBtnClose.bValue = TRUE) THEN
					eOutShutterAct	:= PneuActSetExt;

					IF p_eOutShutterStat = PneuActSetExt AND p_eOutShutterStatus = Done THEN
						eOutShutterAct	:= PneuActIdle;

						tyP0922InletNOutletShutter.tyOutletShutterDC.tyBtnOpen.bRtCompl		:= FALSE;
						tyP0922InletNOutletShutter.tyOutletShutterDC.tyBtnClose.bRtCompl	:= FALSE;
					END_IF

				ELSE
					eOutShutterAct	:= PneuActRstAll;

					IF p_eOutShutterStat = PneuActRstAll AND p_eOutShutterStatus = Done THEN
						eOutShutterAct	:= PneuActIdle;

						tyP0922InletNOutletShutter.tyOutletShutterDC.tyBtnOpen.bRtCompl		:= FALSE;
						tyP0922InletNOutletShutter.tyOutletShutterDC.tyBtnClose.bRtCompl	:= FALSE;
					END_IF

				END_IF
			END_IF
		END_IF

		tyP0922InletNOutletShutter.tyOutletShutterFB.tyBtnOpen.bRtCompl	:= FALSE;
		tyP0922InletNOutletShutter.tyOutletShutterFB.tyBtnOpen.bValue	:= FALSE;
		tyP0922InletNOutletShutter.tyOutletShutterFB.tyBtnClose.bRtCompl:= FALSE;
		tyP0922InletNOutletShutter.tyOutletShutterFB.tyBtnClose.bValue	:= FALSE;

	END_IF

END_ACTION
```

#### Act_OptP0922RstMnl.st
```iecst
ACTION Act_OptP0922RstMnl:

	IF EDGEPOS(p_eInShutterStatus = Error) THEN

		eInShutterAct	:= PneuActIdle;

		tyP0922InletNOutletShutter.tyInletShutterDC.tyBtnClose.bRtCompl	:= FALSE;
		tyP0922InletNOutletShutter.tyInletShutterDC.tyBtnClose.bValue	:= FALSE;
		tyP0922InletNOutletShutter.tyInletShutterDC.tyBtnOpen.bRtCompl	:= FALSE;
		tyP0922InletNOutletShutter.tyInletShutterDC.tyBtnOpen.bValue	:= TRUE;

		tyP0922InletNOutletShutter.tyInletShutterFB.tyBtnClose.bRtCompl	:= FALSE;
		tyP0922InletNOutletShutter.tyInletShutterFB.tyBtnClose.bValue	:= FALSE;
		tyP0922InletNOutletShutter.tyInletShutterFB.tyBtnOpen.bRtCompl	:= FALSE;
		tyP0922InletNOutletShutter.tyInletShutterFB.tyBtnOpen.bValue	:= FALSE;

	END_IF

	IF EDGEPOS(p_eOutShutterStatus = Error) THEN

		eOutShutterAct	:= PneuActIdle;

		tyP0922InletNOutletShutter.tyOutletShutterDC.tyBtnClose.bRtCompl	:= FALSE;
		tyP0922InletNOutletShutter.tyOutletShutterDC.tyBtnClose.bValue		:= FALSE;
		tyP0922InletNOutletShutter.tyOutletShutterDC.tyBtnOpen.bRtCompl		:= FALSE;
		tyP0922InletNOutletShutter.tyOutletShutterDC.tyBtnOpen.bValue		:= FALSE;

		tyP0922InletNOutletShutter.tyOutletShutterFB.tyBtnClose.bRtCompl	:= FALSE;
		tyP0922InletNOutletShutter.tyOutletShutterFB.tyBtnClose.bValue		:= FALSE;
		tyP0922InletNOutletShutter.tyOutletShutterFB.tyBtnOpen.bRtCompl		:= FALSE;
		tyP0922InletNOutletShutter.tyOutletShutterFB.tyBtnOpen.bValue		:= FALSE;

	END_IF

	IF EDGEPOS(bManualMod = FALSE) THEN

		tyP0922InletNOutletShutter.tyInletShutterCom.tyBtnSwitch.bValue		:= FALSE;
		tyP0922InletNOutletShutter.tyOutletShutterCom.tyBtnSwitch.bValue	:= FALSE;

		fUIInRtStatHide(ADR(tyP0922InletNOutletShutter.tyInletShutterDC.tyLyr.uiRtStat));
		fUIInRtStatOff(ADR(tyP0922InletNOutletShutter.tyInletShutterFB.tyLyr.uiRtStat));

		fUIInRtStatHide(ADR(tyP0922InletNOutletShutter.tyOutletShutterDC.tyLyr.uiRtStat));
		fUIInRtStatOff(ADR(tyP0922InletNOutletShutter.tyOutletShutterFB.tyLyr.uiRtStat));

		eInShutterAct	:= PneuActIdle;

		tyP0922InletNOutletShutter.tyInletShutterDC.tyBtnClose.bRtCompl	:= FALSE;
		tyP0922InletNOutletShutter.tyInletShutterDC.tyBtnClose.bValue	:= FALSE;
		tyP0922InletNOutletShutter.tyInletShutterDC.tyBtnOpen.bRtCompl	:= FALSE;
		tyP0922InletNOutletShutter.tyInletShutterDC.tyBtnOpen.bValue	:= TRUE;

		tyP0922InletNOutletShutter.tyInletShutterFB.tyBtnClose.bRtCompl	:= FALSE;
		tyP0922InletNOutletShutter.tyInletShutterFB.tyBtnClose.bValue	:= FALSE;
		tyP0922InletNOutletShutter.tyInletShutterFB.tyBtnOpen.bRtCompl	:= FALSE;
		tyP0922InletNOutletShutter.tyInletShutterFB.tyBtnOpen.bValue	:= FALSE;

		eOutShutterAct	:= PneuActIdle;

		tyP0922InletNOutletShutter.tyOutletShutterDC.tyBtnClose.bRtCompl	:= FALSE;
		tyP0922InletNOutletShutter.tyOutletShutterDC.tyBtnClose.bValue		:= FALSE;
		tyP0922InletNOutletShutter.tyOutletShutterDC.tyBtnOpen.bRtCompl		:= FALSE;
		tyP0922InletNOutletShutter.tyOutletShutterDC.tyBtnOpen.bValue		:= FALSE;

		tyP0922InletNOutletShutter.tyOutletShutterFB.tyBtnClose.bRtCompl	:= FALSE;
		tyP0922InletNOutletShutter.tyOutletShutterFB.tyBtnClose.bValue		:= FALSE;
		tyP0922InletNOutletShutter.tyOutletShutterFB.tyBtnOpen.bRtCompl		:= FALSE;
		tyP0922InletNOutletShutter.tyOutletShutterFB.tyBtnOpen.bValue		:= FALSE;

	END_IF

END_ACTION
```

#### Act_EntP0923Disp.st
```iecst
ACTION Act_EntP0923Disp:

	//Access Address
	p_tyC0002FullMask ACCESS ADR(tyP0923Stopper.tyFullMaskHide);

	p_tyC0004Navi ACCESS ADR(tyP0923Stopper.tyNaviBack);

	p_tyC0005Main ACCESS ADR(tyCommon.tyMain);

	p_tyC0007Notif ACCESS ADR(tyCommon.tyNotif);

	p_tyC0008MsgBox ACCESS ADR(tyP0923Stopper.tyMsgBoxHide);

	p_tyC0009Info ACCESS ADR(tyCommon.tyInfo);

	p_tyC0011Loading ACCESS ADR(tyCommon.tyLoading);

	p_tyP0923StopperCom ACCESS ADR(tyP0923Stopper.tyCom);

	p_tyP0923StopperDC ACCESS ADR(tyP0923Stopper.tyDC);

	p_tyP0923StopperFB ACCESS ADR(tyP0923Stopper.tyFB);

	//Display
	IF tyP0923Stopper.tyCom.tyBtnDCCtrl.bValue = TRUE THEN
		fUIInRtStatOff(ADR(tyP0923Stopper.tyDC.tyLyr.uiRtStat));
		fUIInRtStatHide(ADR(tyP0923Stopper.tyFB.tyLyr.uiRtStat));
	ELSE
		fUIInRtStatHide(ADR(tyP0923Stopper.tyDC.tyLyr.uiRtStat));
		fUIInRtStatOff(ADR(tyP0923Stopper.tyFB.tyLyr.uiRtStat));
	END_IF

END_ACTION
```
